# B&R Automation Studio project BenchEDM_AS6 (part 2)

#### TC_IO_AI.st
```iecst
(* Full Analog Input Handler*)
FUNCTION_BLOCK TC_IO_AI

	CASE VarType OF
		TC_IO_ANALOG_TYPE_INT:
		//LOGICAL
			Signal.IOMapping.VarINT					:= IOMapping.VarINT;
			Signal.Vis.Raw							:= INT_TO_LREAL(Signal.IOMapping.VarINT);
			Signal.Vis.IO							:= Par.M*INT_TO_LREAL(Signal.IOMapping.VarINT)+Par.B;
		//SIMULATION
			IF Sim.Active THEN
				Signal.Vis.IO						:= Sim.Logical;
				IF Par.M <> 0 THEN
					Signal.Vis.Raw					:= (Signal.Vis.IO-Par.B)/Par.M;
					Signal.IOMapping.VarINT			:= LREAL_TO_INT(Signal.Vis.Raw);
				ELSE
					Signal.Vis.Raw					:= 0.0;
					Signal.IOMapping.VarINT			:= 0;
				END_IF;
			END_IF;
		TC_IO_ANALOG_TYPE_USINT:
		//LOGICAL
			Signal.IOMapping.VarUSINT				:= IOMapping.VarUSINT;
			Signal.Vis.Raw							:= USINT_TO_LREAL(Signal.IOMapping.VarUSINT);
			Signal.Vis.IO							:= Par.M*USINT_TO_LREAL(Signal.IOMapping.VarUSINT)+Par.B;
		//SIMULATION
			IF Sim.Active THEN
				Signal.Vis.IO						:= Sim.Logical;
				IF Par.M <> 0 THEN
					Signal.Vis.Raw					:= (Signal.Vis.IO-Par.B)/Par.M;
					Signal.IOMapping.VarUSINT		:= LREAL_TO_USINT(Signal.Vis.Raw);
				ELSE
					Signal.Vis.Raw					:= 0.0;
					Signal.IOMapping.VarUSINT		:= 0;
				END_IF;
			END_IF;
		TC_IO_ANALOG_TYPE_SINT:
		//LOGICAL
			Signal.IOMapping.VarSINT				:= IOMapping.VarSINT;
			Signal.Vis.Raw							:= SINT_TO_LREAL(Signal.IOMapping.VarSINT);
			Signal.Vis.IO							:= Par.M*SINT_TO_LREAL(Signal.IOMapping.VarSINT)+Par.B;
		//SIMULATION
			IF Sim.Active THEN
				Signal.Vis.IO						:= Sim.Logical;
				IF Par.M <> 0 THEN
					Signal.Vis.Raw					:= (Signal.Vis.IO-Par.B)/Par.M;
					Signal.IOMapping.VarSINT		:= LREAL_TO_SINT(Signal.Vis.Raw);
				ELSE
					Signal.Vis.Raw					:= 0.0;
					Signal.IOMapping.VarSINT		:= 0;
				END_IF;
			END_IF;
		TC_IO_ANALOG_TYPE_UINT:
		//LOGICAL
			Signal.IOMapping.VarUINT				:= IOMapping.VarUINT;
			Signal.Vis.Raw							:= UINT_TO_LREAL(Signal.IOMapping.VarUINT);
			Signal.Vis.IO							:= Par.M*UINT_TO_LREAL(Signal.IOMapping.VarUINT)+Par.B;
		//SIMULATION
			IF Sim.Active THEN
				Signal.Vis.IO						:= Sim.Logical;
				IF Par.M <> 0 THEN
					Signal.Vis.Raw					:= (Signal.Vis.IO-Par.B)/Par.M;
					Signal.IOMapping.VarUINT		:= LREAL_TO_UINT(Signal.Vis.Raw);
				ELSE
					Signal.Vis.Raw					:= 0.0;
					Signal.IOMapping.VarUINT		:= 0;
				END_IF;
			END_IF;
		TC_IO_ANALOG_TYPE_DINT:
		//LOGICAL
			Signal.IOMapping.VarDINT				:= IOMapping.VarDINT;
			Signal.Vis.Raw							:= DINT_TO_LREAL(Signal.IOMapping.VarDINT);
			Signal.Vis.IO							:= Par.M*DINT_TO_LREAL(Signal.IOMapping.VarDINT)+Par.B;
		//SIMULATION
			IF Sim.Active THEN
				Signal.Vis.IO						:= Sim.Logical;
				IF Par.M <> 0 THEN
					Signal.Vis.Raw					:= (Signal.Vis.IO-Par.B)/Par.M;
					Signal.IOMapping.VarDINT		:= LREAL_TO_DINT(Signal.Vis.Raw);
				ELSE
					Signal.Vis.Raw					:= 0.0;
					Signal.IOMapping.VarDINT		:= 0;
				END_IF;
			END_IF;
		TC_IO_ANALOG_TYPE_UDINT:
		//LOGICAL
			Signal.IOMapping.VarUDINT				:= IOMapping.VarUDINT;
			Signal.Vis.Raw							:= UDINT_TO_LREAL(Signal.IOMapping.VarUDINT);
			Signal.Vis.IO							:= Par.M*UDINT_TO_LREAL(Signal.IOMapping.VarUDINT)+Par.B;
		//SIMULATION
			IF Sim.Active THEN
				Signal.Vis.IO						:= Sim.Logical;
				IF Par.M <> 0 THEN
					Signal.Vis.Raw					:= (Signal.Vis.IO-Par.B)/Par.M;
					Signal.IOMapping.VarUDINT		:= LREAL_TO_UDINT(Signal.Vis.Raw);
				ELSE
					Signal.Vis.Raw					:= 0.0;
					Signal.IOMapping.VarUDINT		:= 0;
				END_IF;
			END_IF;
		TC_IO_ANALOG_TYPE_REAL:
		//LOGICAL
			Signal.IOMapping.VarREAL				:= IOMapping.VarREAL;
			Signal.Vis.Raw							:= REAL_TO_LREAL(Signal.IOMapping.VarREAL);
			Signal.Vis.IO							:= Par.M*REAL_TO_LREAL(Signal.IOMapping.VarREAL)+Par.B;
		//SIMULATION
			IF Sim.Active THEN
				Signal.Vis.IO						:= Sim.Logical;
				IF Par.M <> 0 THEN
					Signal.Vis.Raw					:= (Signal.Vis.IO-Par.B)/Par.M;
					Signal.IOMapping.VarREAL		:= LREAL_TO_REAL(Signal.Vis.Raw);
				ELSE
					Signal.Vis.Raw					:= 0.0;
					Signal.IOMapping.VarREAL		:= 0;
				END_IF;
			END_IF;
		TC_IO_ANALOG_TYPE_LREAL:
		//LOGICAL
			Signal.IOMapping.VarLREAL				:= IOMapping.VarLREAL;
			Signal.Vis.Raw							:= Signal.IOMapping.VarLREAL;
			Signal.Vis.IO							:= Par.M*Signal.IOMapping.VarLREAL+Par.B;
		//SIMULATION
			IF Sim.Active THEN
				Signal.Vis.IO						:= Sim.Logical;
				IF Par.M <> 0 THEN
					Signal.Vis.Raw					:= (Signal.Vis.IO-Par.B)/Par.M;
					Signal.IOMapping.VarLREAL		:= Signal.Vis.Raw;
				ELSE
					Signal.Vis.Raw					:= 0.0;
					Signal.IOMapping.VarLREAL		:= 0;
				END_IF;
			END_IF;
	END_CASE;
	Signal.Logical									:= Signal.Vis.IO;
//FORCING
	IF Forcing.On XOR Forcing.Off THEN
		IF Forcing.Off THEN
			Signal.Logical							:= 0.0;
		ELSIF Forcing.On THEN
			Signal.Logical							:= Forcing.Value;
		END_IF;
	END_IF;
//LIMITING
	Signal.UnlimitedLogical							:= Signal.Logical;
	Signal.MaxExceeded								:= FALSE;
	IF Signal.Logical > Par.MaxValue THEN
		Signal.MaxExceeded							:= TRUE;
		Signal.Logical								:= Par.MaxValue;
	END_IF;
	Signal.MinExceeded								:= FALSE;
	IF Signal.Logical < Par.MinValue THEN
		Signal.MinExceeded							:= TRUE;
		Signal.Logical								:= Par.MinValue;
	END_IF;
//FILTERING
	Internal.Filter 								:= Par.Filter;
	IF Par.Filter < 0.0 THEN
		Internal.Filter 							:= 0.0;
	ELSIF Internal.Filter > 1.0 THEN
		Internal.Filter 							:= 0.99999999;
	END_IF;
	IF NOT Internal.InitFilter OR Internal.LastFilter <> Internal.Filter THEN
		Internal.InitFilter							:= TRUE;
		Internal.LastFilter 						:= Internal.Filter;
		Signal.Filtered 							:= Signal.Logical;
	ELSE
		Signal.Filtered 							:= Signal.Logical*(1.0-Internal.Filter) + Signal.Filtered*Internal.Filter;
	END_IF;
	IF Signal.Filtered > Par.MaxValue THEN
		Signal.Filtered 							:= Par.MaxValue;
	ELSIF Signal.Filtered < Par.MinValue THEN
		Signal.Filtered 							:= Par.MinValue;
	END_IF;
	Signal.Vis.App									:= Signal.Filtered;
END_FUNCTION_BLOCK
```

### Library Logical/Libraries/TC_Dir (IEC)
Depends on: TC_General, AsBrStr, standard, brsystem, FileIO, AsUSB, astime

#### Types.typ - Exported data types
```iecst
TYPE
	TC_DirDef_Sanitize_typ : 	STRUCT
		AllowUndefinedDir : BOOL;
		SanitizeFilesByExt : BOOL;
		SanitizeFilesByRoot : BOOL;
		FileExtension : STRING[260];
		FileRoot : STRING[260];
		MaxSize : UDINT;
		MaxFiles : UDINT;
	END_STRUCT;
	TC_DirDef_typ : 	STRUCT
		Valid : BOOL;
		DirPath : STRING[260];
		Sanitize : TC_DirDef_Sanitize_typ;
	END_STRUCT;
	TC_DirMake_Internal_typ : 	STRUCT
		State : TC_DIRMAKE_STATE_ENUM;
		DirDefItem : TC_DirDef_typ;
		DirCreate_0 : DirCreate;
		DirIdx : INT;
	END_STRUCT;
	TC_DIRMAKE_STATE_ENUM :
		(
		DIRMAKE_RESET,
		DIRMAKE_IDLE,
		DIRMAKE_CREATE_CMD,
		DIRMAKE_CREATE_WAIT,
		DIRMAKE_DONE,
		DIRMAKE_ERROR
		);
	TC_DirReadAll_Internal_typ : 	STRUCT
		State : TC_DIRREADALL_STATE_ENUM;
		DirOpen_0 : DirOpen;
		DirReadEx_0 : DirReadEx;
		DirClose_0 : DirClose;
		i : INT;
		FileListIdx : INT;
		DirIdent : UDINT;
		DirData : fiDIR_READ_EX_DATA;
		FileListItem : TC_FileList_typ;
		CurrentDirPath : STRING[260];
	END_STRUCT;
	TC_DIRREADALL_STATE_ENUM :
		(
		DIRREADALL_RESET,
		DIRREADALL_IDLE,
		DIRREADALL_OPEN_CMD,
		DIRREADALL_OPEN_WAIT,
		DIRREADALL_READ_CMD,
		DIRREADALL_READ_WAIT,
		DIRREADALL_CLOSE_WAIT,
		DIRREADALL_EVALUATE,
		DIRREADALL_DONE,
		DIRREADALL_ERROR
		);
	TC_DirSanitize_Internal_typ : 	STRUCT
		State : TC_DIRSANITIZE_STATE_ENUM;
		DirDeleteEx_0 : DirDeleteEx;
		FileDelete_0 : FileDelete;
		DirDefItem : TC_DirDef_typ;
		FileListItem : TC_FileList_typ;
		FileListItem1 : TC_FileList_typ;
		i : INT;
		j : INT;
		FileListIdx : INT;
		Size : UDINT;
		DirIdent : UDINT;
		SizeCount : UDINT;
		FileCount : UDINT;
		DirData : fiDIR_READ_EX_DATA;
		Found : BOOL;
		Find : INT;
		TempPath : STRING[260];
		CurrentDirIdx : INT;
	END_STRUCT;
	TC_DIRSANITIZE_STATE_ENUM :
		(
		DIRSANITIZE_RESET,
		DIRSANITIZE_IDLE,
		DIRSANITIZE_EVALUATE_DIR,
		DIRSANITIZE_DELETE_DIR_CMD,
		DIRSANITIZE_DELETE_DIR_WAIT,
		DIRSANITIZE_DELETE_DIR_PROCESS,
		DIRSANITIZE_EVALUATE_FILE,
		DIRSANITIZE_DELETE_FILE_CMD,
		DIRSANITIZE_DELETE_FILE_WAIT,
		DIRSANITIZE_DONE,
		DIRSANITIZE_ERROR
		);
	TC_Dir_Transfer_Internal_typ : 	STRUCT
		State : TC_DIR_TRANSFER_STATE_ENUM;
		TransferListItem : TC_Dir_Transfer_List_typ;
		ListIdx : INT;
		DirCopy_0 : DirCopy;
		FileCopy_0 : FileCopy;
		DirDeleteEx_0 : DirDeleteEx;
		DirCreate_0 : DirCreate;
		FileDelete_0 : FileDelete;
	END_STRUCT;
	TC_Dir_Transfer_List_typ : 	STRUCT
		Valid : BOOL;
		SrcOrDestUSB : BOOL;
		IsDir : BOOL;
		SrcDelete : BOOL;
		SrcCreateDir : BOOL;
		NoTransfer : BOOL;
		SrcDev : STRING[80];
		SrcPath : STRING[260];
		DestDev : STRING[80];
		DestPath : STRING[260];
	END_STRUCT;
	TC_DIR_TRANSFER_STATE_ENUM :
		(
		TRANSFER_RESET,
		TRANSFER_IDLE,
		TRANSFER_CHECK_LIST,
		TRANSFER_DIR_COPY_CMD,
		TRANSFER_DIR_COPY_WAIT,
		TRANSFER_FILE_COPY_CMD,
		TRANSFER_FILE_COPY_WAIT,
		TRANSFER_DIR_DELETE_CMD,
		TRANSFER_DIR_DELETE_WAIT,
		TRANSFER_FILE_DELETE_CMD,
		TRANSFER_FILE_DELETE_WAIT,
		TRANSFER_DIR_CREATE_CMD,
		TRANSFER_DIR_CREATE_WAIT,
		TRANSFER_DONE,
		TRANSFER_ERROR
		);
	TC_Dir_USB_Connect_Internal_typ : 	STRUCT
		UsbNodeListGet_0 : UsbNodeListGet;
		UsbNodeGet_0 : UsbNodeGet;
		DevLink_0 : DevLink;
		UsbMsDeviceReady_0 : UsbMsDeviceReady;
		DevUnlink_0 : DevUnlink;
		CTON_Delay : CTON;
		NodeList : UDINT;
		Node : usbNode_typ;
		ParString : STRING[1000];
		Handle : UDINT;
		State : TC_USB_CONNECT_STATE_ENUM;
	END_STRUCT;
	TC_FileList_typ : 	STRUCT
		Path : STRING[260];
		DateUDINT : UDINT;
		Size : UDINT;
		IsDir : BOOL;
		DirIdx : INT;
		Internal : USINT; (*0=unread, 1=delete, 2=parentDirDelete, 3=remove*)
	END_STRUCT;
	TC_USB_CONNECT_STATE_ENUM :
		(
		USB_CONNECT_RESET,
		USB_CONNECT_IDLE,
		USB_CONNECT_GET_LIST_CMD,
		USB_CONNECT_GET_LIST_WAIT,
		USB_CONNECT_GET_NODE_CMD,
		USB_CONNECT_GET_NODE_WAIT,
		USB_CONNECT_DEVLINK_CMD,
		USB_CONNECT_DEVLINK_WAIT,
		USB_CONNECT_CHECK_CONNECTED,
		USB_CONNECT_CONNECTED,
		USB_CONNECT_DEVUNLINK_CMD,
		USB_CONNECT_DEVUNLINK_WAIT,
		USB_CONNECT_DELAY,
		USB_CONNECT_DONE,
		USB_CONNECT_ERROR
		);
END_TYPE
```

#### TC_Dir.fun - Exported functions and function blocks
```iecst
{REDUND_ERROR} FUNCTION_BLOCK TC_DirMake (* *) (*$GROUP=User,$CAT=User,$GROUPICON=User.png,$CATICON=User.png*)
	VAR_INPUT
		enable : BOOL;
		pDevice : UDINT;
		pDirDef : UDINT;
	END_VAR
	VAR_OUTPUT
		status : UINT;
	END_VAR
	VAR
		Internal : TC_DirMake_Internal_typ;
	END_VAR
END_FUNCTION_BLOCK

{REDUND_ERROR} FUNCTION_BLOCK TC_DirReadAll (*Reads Entire File Device*) (*$GROUP=User,$CAT=User,$GROUPICON=User.png,$CATICON=User.png*)
	VAR_INPUT
		enable : BOOL;
		pDevice : UDINT;
		pFileList : UDINT;
	END_VAR
	VAR_OUTPUT
		status : UINT;
	END_VAR
	VAR
		Internal : TC_DirReadAll_Internal_typ;
	END_VAR
END_FUNCTION_BLOCK

{REDUND_ERROR} FUNCTION_BLOCK TC_DirSanitize (*Sanitizes File Device*) (*$GROUP=User,$CAT=User,$GROUPICON=User.png,$CATICON=User.png*)
	VAR_INPUT
		enable : BOOL;
		pDevice : UDINT;
		pDirDef : UDINT;
		pFileList : UDINT;
	END_VAR
	VAR_OUTPUT
		status : UINT;
	END_VAR
	VAR
		Internal : TC_DirSanitize_Internal_typ;
	END_VAR
END_FUNCTION_BLOCK

{REDUND_ERROR} FUNCTION_BLOCK TC_Dir_USB_Connect (*TODO: Add your comment here*) (*$GROUP=User,$CAT=User,$GROUPICON=User.png,$CATICON=User.png*)
	VAR_INPUT
		enable : BOOL;
		reset : BOOL;
		refresh : BOOL;
		delay : REAL;
	END_VAR
	VAR_OUTPUT
		status : UINT;
		connected : BOOL;
	END_VAR
	VAR
		Internal : TC_Dir_USB_Connect_Internal_typ;
	END_VAR
END_FUNCTION_BLOCK

{REDUND_ERROR} FUNCTION_BLOCK TC_Dir_Transfer (*Transfer List from Device to Another*) (*$GROUP=User,$CAT=User,$GROUPICON=User.png,$CATICON=User.png*)
	VAR_INPUT
		enable : BOOL;
		USB_Connected : BOOL;
		pTransferList : UDINT;
	END_VAR
	VAR_OUTPUT
		index : INT;
		status : UINT;
	END_VAR
	VAR
		Internal : TC_Dir_Transfer_Internal_typ;
	END_VAR
END_FUNCTION_BLOCK
```

#### TC_DirMake.st
```iecst
FUNCTION_BLOCK TC_DirMake

	IF enable = FALSE THEN
		Internal.State									:= DIRMAKE_RESET;
	END_IF;

	CASE Internal.State OF
		DIRMAKE_RESET:
			status										:= 65534;
			brsmemset(ADR(Internal),0,SIZEOF(Internal));
			Internal.State								:= DIRMAKE_IDLE;
		DIRMAKE_IDLE:
			status										:= 65534;
			IF enable THEN
				IF pDevice <> 0 AND pDirDef <> 0 THEN
					status								:= 65535;
					brsmemset(ADR(Internal),0,SIZEOF(Internal));
					Internal.State						:= DIRMAKE_CREATE_CMD;
				ELSE
					status								:= 60001;
					Internal.State						:= DIRMAKE_ERROR;
				END_IF;
			END_IF;
		DIRMAKE_CREATE_CMD:
			status										:= 65535;
			IF Internal.DirIdx >= 0 AND Internal.DirIdx <= MAX_DIR_DEF_IDX THEN
				brsmemcpy(ADR(Internal.DirDefItem),pDirDef+SIZEOF(Internal.DirDefItem)*Internal.DirIdx,SIZEOF(Internal.DirDefItem));
				IF Internal.DirDefItem.Valid THEN
					IF Internal.DirDefItem.DirPath <> '' AND Internal.DirDefItem.DirPath <> '/' THEN
						Internal.DirCreate_0.enable 	:= TRUE;
						Internal.DirCreate_0.pDevice	:= pDevice;
						Internal.DirCreate_0.pName		:= ADR(Internal.DirDefItem.DirPath);
						Internal.State					:= DIRMAKE_CREATE_WAIT;
					ELSE
						Internal.DirIdx 				:= Internal.DirIdx + 1;
					END_IF;
				ELSE
					Internal.State						:= DIRMAKE_DONE;
				END_IF;
			ELSE
				Internal.State							:= DIRMAKE_DONE;
			END_IF;
		DIRMAKE_CREATE_WAIT:
			status										:= 65535;
			IF Internal.DirCreate_0.status = ERR_OK OR Internal.DirCreate_0.status = fiERR_DIR_ALREADY_EXIST THEN
				Internal.DirCreate_0.enable 			:= FALSE;
				Internal.DirIdx 						:= Internal.DirIdx + 1;
				Internal.State 							:= DIRMAKE_CREATE_CMD;
			ELSIF Internal.DirCreate_0.status <> ERR_FUB_BUSY AND Internal.DirCreate_0.status <> ERR_FUB_ENABLE_FALSE THEN
				Internal.DirCreate_0.enable 			:= FALSE;
				status									:= Internal.DirCreate_0.status;
				Internal.State 							:= DIRMAKE_ERROR;
			END_IF;
		DIRMAKE_DONE:
			status										:= 0;
		DIRMAKE_ERROR:
			// Error
	END_CASE;
	Internal.DirCreate_0();

END_FUNCTION_BLOCK
```

#### TC_DirSanitize.st
```iecst
(* Sanitizes File Device *)
FUNCTION_BLOCK TC_DirSanitize
	IF enable = FALSE THEN
		Internal.State										:= DIRSANITIZE_RESET;
	END_IF;

	CASE Internal.State OF
		DIRSANITIZE_RESET:
			status											:= 65534;
			brsmemset(ADR(Internal),0,SIZEOF(Internal));
			Internal.State									:= DIRSANITIZE_IDLE;
		DIRSANITIZE_IDLE:
			status											:= 65534;
			IF enable THEN
				IF pDevice <> 0 AND pDirDef <> 0 AND pFileList <> 0 THEN
					brsmemset(ADR(Internal),0,SIZEOF(Internal));
					status									:= 65535;
					Internal.State							:= DIRSANITIZE_EVALUATE_DIR;
				ELSE
					brsmemset(ADR(Internal),0,SIZEOF(Internal));
					status									:= 60001;
					Internal.State							:= DIRSANITIZE_ERROR;
				END_IF;
			END_IF;
		DIRSANITIZE_EVALUATE_DIR:
			status											:= 65535;
			// Determine DirIdx
			FOR Internal.i := 0 TO MAX_DIR_MAN_FILE_LIST_IDX DO
				brsmemcpy(ADR(Internal.FileListItem),pFileList+SIZEOF(Internal.FileListItem)*Internal.i,SIZEOF(Internal.FileListItem));
				IF Internal.FileListItem.Path = '' AND Internal.FileListItem.IsDir = FALSE THEN
					EXIT;
				ELSE
					Internal.Found 							:= FALSE;
					FOR Internal.j := 0 TO MAX_DIR_DEF_IDX DO
						brsmemcpy(ADR(Internal.DirDefItem),pDirDef+SIZEOF(Internal.DirDefItem)*Internal.j,SIZEOF(Internal.DirDefItem));
						IF Internal.DirDefItem.Valid THEN
							IF Internal.FileListItem.Path = Internal.DirDefItem.DirPath OR Internal.FileListItem.Path = '' THEN
								Internal.FileListItem.DirIdx := Internal.j;
								Internal.Found 				:= TRUE;
								EXIT;
							END_IF;
						END_IF;
					END_FOR;
					IF NOT Internal.Found THEN
						FOR Internal.j := MAX_DIR_DEF_IDX TO 0 BY -1 DO
							brsmemcpy(ADR(Internal.DirDefItem),pDirDef+SIZEOF(Internal.DirDefItem)*Internal.j,SIZEOF(Internal.DirDefItem));
							IF Internal.DirDefItem.Valid THEN
								Internal.Find := FIND(Internal.FileListItem.Path,Internal.DirDefItem.DirPath);
								IF Internal.Find <> 0 THEN
									Internal.TempPath := DELETE(Internal.FileListItem.Path,LEN(Internal.DirDefItem.DirPath),1);
									IF FIND(Internal.TempPath,'/') <> 0 OR Internal.DirDefItem.DirPath = '' THEN
										Internal.FileListItem.DirIdx := Internal.j;
										EXIT;
									END_IF;
								END_IF;
							END_IF;
						END_FOR;
					END_IF;
					brsmemcpy(pFileList+SIZEOF(Internal.FileListItem)*Internal.i,ADR(Internal.FileListItem),SIZEOF(Internal.FileListItem));
				END_IF;
			END_FOR;

			// Handle Directory Sanitation
			Internal.Found									:= FALSE;
			FOR Internal.i := 0 TO MAX_DIR_MAN_FILE_LIST_IDX DO
				brsmemcpy(ADR(Internal.FileListItem),pFileList+SIZEOF(Internal.FileListItem)*Internal.i,SIZEOF(Internal.FileListItem));
				IF Internal.FileListItem.Path = '' AND Internal.FileListItem.IsDir = FALSE THEN
					EXIT;
				ELSIF Internal.FileListItem.IsDir THEN
					brsmemcpy(ADR(Internal.DirDefItem),pDirDef+SIZEOF(Internal.DirDefItem)*Internal.FileListItem.DirIdx,SIZEOF(Internal.DirDefItem));
					IF NOT Internal.DirDefItem.Sanitize.AllowUndefinedDir AND Internal.DirDefItem.DirPath <> Internal.FileListItem.Path THEN
						Internal.Found					:= TRUE;
						Internal.FileListItem.Internal.1 := 1;
						brsmemcpy(pFileList+SIZEOF(Internal.FileListItem)*Internal.i,ADR(Internal.FileListItem),SIZEOF(Internal.FileListItem));
					END_IF;
				END_IF;
			END_FOR;
			Internal.State 									:= DIRSANITIZE_DELETE_DIR_CMD;
		DIRSANITIZE_DELETE_DIR_CMD:
			status											:= 65535;
			Internal.Found									:= FALSE;
			FOR Internal.i := 0 TO MAX_DIR_MAN_FILE_LIST_IDX DO
				brsmemcpy(ADR(Internal.FileListItem),pFileList+SIZEOF(Internal.FileListItem)*Internal.i,SIZEOF(Internal.FileListItem));
				IF Internal.FileListItem.Path = '' AND Internal.FileListItem.IsDir = FALSE THEN
					EXIT;
				ELSIF Internal.FileListItem.IsDir AND Internal.FileListItem.Internal.1 = 1 AND NOT Internal.FileListItem.Internal.2 = 1 THEN
					Internal.Found							:= TRUE;
					EXIT;
				END_IF;
			END_FOR;
			IF Internal.Found THEN
				Internal.DirDeleteEx_0.enable 				:= TRUE;
				Internal.DirDeleteEx_0.pDevice 				:= pDevice;
				Internal.DirDeleteEx_0.pName 				:= ADR(Internal.FileListItem.Path);
				Internal.State 								:= DIRSANITIZE_DELETE_DIR_WAIT;
			ELSE
				Internal.State 								:= DIRSANITIZE_EVALUATE_FILE;
			END_IF;
		DIRSANITIZE_DELETE_DIR_WAIT:
			status											:= 65535;
			IF Internal.DirDeleteEx_0.status = 0 OR (Internal.DirDeleteEx_0.status <> ERR_FUB_BUSY AND Internal.DirDeleteEx_0.status <> ERR_FUB_ENABLE_FALSE) THEN
				Internal.DirDeleteEx_0.enable 				:= FALSE;
				Internal.FileListItem1 						:= Internal.FileListItem;
				FOR Internal.i := 0 TO MAX_DIR_MAN_FILE_LIST_IDX DO
					brsmemcpy(ADR(Internal.FileListItem),pFileList+SIZEOF(Internal.FileListItem)*Internal.i,SIZEOF(Internal.FileListItem));
					IF Internal.FileListItem.Path = '' AND Internal.FileListItem.IsDir = FALSE THEN
						EXIT;
					ELSIF FIND(Internal.FileListItem.Path,Internal.FileListItem1.Path) <> 0 THEN
						Internal.FileListItem.Internal.3 	:= 1;
						brsmemcpy(pFileList+SIZEOF(Internal.FileListItem)*Internal.i,ADR(Internal.FileListItem),SIZEOF(Internal.FileListItem));
					END_IF;
				END_FOR;
				Internal.j 									:= 0;
				FOR Internal.i := 0 TO MAX_DIR_MAN_FILE_LIST_IDX DO
					brsmemcpy(ADR(Internal.FileListItem),pFileList+SIZEOF(Internal.FileListItem)*Internal.i,SIZEOF(Internal.FileListItem));
					IF Internal.FileListItem.Path = '' AND Internal.FileListItem.IsDir = FALSE THEN
						EXIT;
					ELSIF Internal.FileListItem.Internal.3 = 0 THEN
						IF Internal.j <> Internal.i THEN
							Internal.Size						:= (MAX_DIR_MAN_FILE_LIST_IDX+1-Internal.i);
							brsmemmove(pFileList+Internal.j*SIZEOF(Internal.FileListItem),pFileList+Internal.i*SIZEOF(Internal.FileListItem),SIZEOF(Internal.FileListItem)*Internal.Size);
							brsmemset(pFileList+(Internal.j+Internal.Size)*SIZEOF(Internal.FileListItem),0,SIZEOF(Internal.FileListItem)*(Internal.i-Internal.j));
						END_IF;
						Internal.j							:= Internal.j + (Internal.i-Internal.j)+1;
						Internal.i							:= Internal.j-1;
					ELSE
						brsmemset(pFileList+Internal.i*SIZEOF(Internal.FileListItem),0,SIZEOF(Internal.FileListItem));
					END_IF;
				END_FOR;
				Internal.State 								:= DIRSANITIZE_DELETE_DIR_CMD;
			END_IF;
		DIRSANITIZE_EVALUATE_FILE:
			status											:= 65535;

			// Handle File Sanitation By Root
			Internal.Found									:= FALSE;
			FOR Internal.i := 0 TO MAX_DIR_MAN_FILE_LIST_IDX DO
				brsmemcpy(ADR(Internal.FileListItem),pFileList+SIZEOF(Internal.FileListItem)*Internal.i,SIZEOF(Internal.FileListItem));
				IF Internal.FileListItem.Path = '' AND Internal.FileListItem.IsDir = FALSE THEN
					EXIT;
				ELSIF NOT Internal.FileListItem.IsDir THEN
					brsmemcpy(ADR(Internal.DirDefItem),pDirDef+SIZEOF(Internal.DirDefItem)*Internal.FileListItem.DirIdx,SIZEOF(Internal.DirDefItem));
					IF Internal.DirDefItem.Sanitize.SanitizeFilesByRoot THEN
						Internal.TempPath 					:= '';
						brsstrcat(ADR(Internal.TempPath),ADR(Internal.DirDefItem.DirPath));
						brsstrcat(ADR(Internal.TempPath),ADR('/'));
						brsstrcat(ADR(Internal.TempPath),ADR(Internal.DirDefItem.Sanitize.FileRoot));
						IF FIND(Internal.FileListItem.Path,Internal.TempPath) = 0 THEN
							Internal.Found					:= TRUE;
							Internal.FileListItem.Internal.1 := 1;
							brsmemcpy(pFileList+SIZEOF(Internal.FileListItem)*Internal.i,ADR(Internal.FileListItem),SIZEOF(Internal.FileListItem));
						END_IF;
					END_IF;
					IF Internal.DirDefItem.Sanitize.SanitizeFilesByExt THEN
						IF FIND(Internal.FileListItem.Path,Internal.DirDefItem.Sanitize.FileExtension) = 0 THEN
							Internal.Found					:= TRUE;
							Internal.FileListItem.Internal.1 := 1;
							brsmemcpy(pFileList+SIZEOF(Internal.FileListItem)*Internal.i,ADR(Internal.FileListItem),SIZEOF(Internal.FileListItem));
						END_IF;
					END_IF;
				END_IF;
			END_FOR;

			// Check if found in the last step. If so we have to go delete these files before counting them for size and number of files.
			IF Internal.Found THEN
				Internal.State 								:= DIRSANITIZE_DELETE_FILE_CMD;
			ELSE
				// Reorder Files for Evaluation
				FOR Internal.i := 0 TO MAX_DIR_MAN_FILE_LIST_IDX-1 DO
					brsmemcpy(ADR(Internal.FileListItem),pFileList+SIZEOF(Internal.FileListItem)*Internal.i,SIZEOF(Internal.FileListItem));
					brsmemcpy(ADR(Internal.FileListItem1),pFileList+SIZEOF(Internal.FileListItem1)*(Internal.i+1),SIZEOF(Internal.FileListItem1));
					IF (Internal.FileListItem.Path = '' AND Internal.FileListItem.IsDir = FALSE) OR (Internal.FileListItem1.Path = '' AND Internal.FileListItem1.IsDir = FALSE) THEN
						EXIT;
					ELSE
						IF Internal.FileListItem.DirIdx = Internal.FileListItem1.DirIdx THEN
							IF Internal.FileListItem.DateUDINT < Internal.FileListItem1.DateUDINT THEN
								brsmemcpy(pFileList+SIZEOF(Internal.FileListItem1)*Internal.i,ADR(Internal.FileListItem1),SIZEOF(Internal.FileListItem1));
								brsmemcpy(pFileList+SIZEOF(Internal.FileListItem)*(Internal.i+1),ADR(Internal.FileListItem),SIZEOF(Internal.FileListItem));
							END_IF;
						END_IF;
					END_IF;
				END_FOR;
				// Delete Files Based On File Number and Size Restriction
				Internal.Found								:= FALSE;
				Internal.CurrentDirIdx						:= 0;
				Internal.FileCount							:= 1;
				Internal.SizeCount							:= 0;
				FOR Internal.i := 0 TO MAX_DIR_MAN_FILE_LIST_IDX DO
					brsmemcpy(ADR(Internal.FileListItem),pFileList+SIZEOF(Internal.FileListItem)*Internal.i,SIZEOF(Internal.FileListItem));
					IF Internal.FileListItem.Path = '' AND Internal.FileListItem.IsDir = FALSE THEN
						EXIT;
					ELSIF NOT Internal.FileListItem.IsDir THEN
						IF Internal.CurrentDirIdx <> Internal.FileListItem.DirIdx THEN
							Internal.CurrentDirIdx 			:= Internal.FileListItem.DirIdx;
							Internal.FileCount				:= 1;
							Internal.SizeCount				:= Internal.FileListItem.Size;
						ELSE
							Internal.FileCount				:= Internal.FileCount + 1;
							Internal.SizeCount				:= Internal.SizeCount + Internal.FileListItem.Size;
						END_IF;
						brsmemcpy(ADR(Internal.DirDefItem),pDirDef+SIZEOF(Internal.DirDefItem)*Internal.FileListItem.DirIdx,SIZEOF(Internal.DirDefItem));
						IF Internal.FileCount > Internal.DirDefItem.Sanitize.MaxFiles OR Internal.SizeCount > Internal.DirDefItem.Sanitize.MaxSize THEN
							Internal.Found					:= TRUE;
							Internal.FileListItem.Internal.1 := 1;
							brsmemcpy(pFileList+SIZEOF(Internal.FileListItem)*Internal.i,ADR(Internal.FileListItem),SIZEOF(Internal.FileListItem));
						END_IF;
					END_IF;
				END_FOR;
				IF Internal.Found THEN
					Internal.State 							:= DIRSANITIZE_DELETE_FILE_CMD;
				ELSE
					Internal.State 							:= DIRSANITIZE_DONE;
				END_IF;
			END_IF;
		DIRSANITIZE_DELETE_FILE_CMD:
			status											:= 65535;
			Internal.Found									:= FALSE;
			FOR Internal.i := 0 TO MAX_DIR_MAN_FILE_LIST_IDX DO
				brsmemcpy(ADR(Internal.FileListItem),pFileList+SIZEOF(Internal.FileListItem)*Internal.i,SIZEOF(Internal.FileListItem));
				IF Internal.FileListItem.Path = '' AND Internal.FileListItem.IsDir = FALSE THEN
					EXIT;
				ELSIF NOT Internal.FileListItem.IsDir AND Internal.FileListItem.Internal.1 = 1 THEN
					Internal.FileListItem.Internal.1 := 0;
					Internal.FileListItem.Internal.3 := 1;
					brsmemcpy(pFileList+SIZEOF(Internal.FileListItem)*Internal.i,ADR(Internal.FileListItem),SIZEOF(Internal.FileListItem));
					Internal.Found							:= TRUE;
					EXIT;
				END_IF;
			END_FOR;
			IF Internal.Found THEN
				Internal.FileDelete_0.enable 				:= TRUE;
				Internal.FileDelete_0.pDevice 				:= pDevice;
				Internal.FileDelete_0.pName 				:= ADR(Internal.FileListItem.Path);
				Internal.State 								:= DIRSANITIZE_DELETE_FILE_WAIT;
			ELSE
				Internal.State 								:= DIRSANITIZE_EVALUATE_FILE;
			END_IF;
		DIRSANITIZE_DELETE_FILE_WAIT:
			status											:= 65535;
			IF Internal.FileDelete_0.status = 0 OR (Internal.FileDelete_0.status <> ERR_FUB_BUSY AND Internal.FileDelete_0.status <> ERR_FUB_ENABLE_FALSE) THEN
				Internal.FileDelete_0.enable 				:= FALSE;
				Internal.j 									:= 0;
				FOR Internal.i := 0 TO MAX_DIR_MAN_FILE_LIST_IDX DO
					brsmemcpy(ADR(Internal.FileListItem),pFileList+SIZEOF(Internal.FileListItem)*Internal.i,SIZEOF(Internal.FileListItem));
					IF Internal.FileListItem.Path = '' AND Internal.FileListItem.IsDir = FALSE THEN
						EXIT;
					ELSIF Internal.FileListItem.Internal.3 = 0 THEN
						IF Internal.j <> Internal.i THEN
							Internal.Size						:= (MAX_DIR_MAN_FILE_LIST_IDX+1-Internal.i);
							brsmemmove(pFileList+Internal.j*SIZEOF(Internal.FileListItem),pFileList+Internal.i*SIZEOF(Internal.FileListItem),SIZEOF(Internal.FileListItem)*Internal.Size);
							brsmemset(pFileList+(Internal.j+Internal.Size)*SIZEOF(Internal.FileListItem),0,SIZEOF(Internal.FileListItem)*(Internal.i-Internal.j));
						END_IF;
						Internal.j							:= Internal.j + (Internal.i-Internal.j)+1;
						Internal.i							:= Internal.j-1;
					ELSE
						brsmemset(pFileList+Internal.i*SIZEOF(Internal.FileListItem),0,SIZEOF(Internal.FileListItem));
					END_IF;
				END_FOR;
				Internal.State 								:= DIRSANITIZE_DELETE_FILE_CMD;
			END_IF;
		DIRSANITIZE_DONE:
			status											:= 0;
		DIRSANITIZE_ERROR:
			// Error
	END_CASE;

	Internal.FileDelete_0();
	Internal.DirDeleteEx_0();

END_FUNCTION_BLOCK
```

#### TC_Dir_USB_Connect.st
```iecst
// This function only supports a single USB flash drive, additional will be ignored.
// When connected the USB can be accessed using Dev Name 'USB_DEVICE'

FUNCTION_BLOCK TC_Dir_USB_Connect

	IF enable = FALSE OR reset THEN
		Internal.State											:= USB_CONNECT_RESET;
	END_IF;

	CASE Internal.State OF
		USB_CONNECT_RESET:
			status												:= 65534;
			brsmemset(ADR(Internal),0,SIZEOF(Internal));
			connected											:= FALSE;
			Internal.State										:= USB_CONNECT_IDLE;
		USB_CONNECT_IDLE:
			status												:= 65534;
			IF enable THEN
				status											:= 65535;
				Internal.State									:= USB_CONNECT_GET_LIST_CMD;
			END_IF;
		USB_CONNECT_GET_LIST_CMD:
			status												:= 65535;
			Internal.UsbNodeListGet_0.enable 					:= TRUE;
			Internal.UsbNodeListGet_0.pBuffer 					:= ADR(Internal.NodeList);
			Internal.UsbNodeListGet_0.bufferSize 				:= SIZEOF(Internal.NodeList);
			Internal.UsbNodeListGet_0.filterInterfaceClass 		:= 8; // FIND ONLY USB FLASH DRIVES
			Internal.UsbNodeListGet_0.filterInterfaceSubClass 	:= 6; // FIND ONLY USB FLASH DRIVES
			Internal.State 										:= USB_CONNECT_GET_LIST_WAIT;
		USB_CONNECT_GET_LIST_WAIT:
			status												:= 65535;
			IF Internal.UsbNodeListGet_0.status = 0 THEN
				Internal.UsbNodeListGet_0.enable 				:= FALSE;
				Internal.State 									:= USB_CONNECT_GET_NODE_CMD;
			ELSIF Internal.UsbNodeListGet_0.status <> ERR_FUB_BUSY AND Internal.UsbNodeListGet_0.status <> ERR_FUB_ENABLE_FALSE THEN
				IF Internal.UsbNodeListGet_0.status <> asusbERR_USB_NOTFOUND THEN
					Internal.UsbNodeListGet_0.enable 			:= FALSE;
					status										:= Internal.UsbNodeListGet_0.status;
					Internal.State 								:= USB_CONNECT_ERROR;
				ELSE
					Internal.UsbNodeListGet_0.enable 			:= FALSE;
					Internal.State 								:= USB_CONNECT_DELAY;
				END_IF;
			END_IF;
		USB_CONNECT_GET_NODE_CMD:
			status												:= 65535;
			Internal.UsbNodeGet_0.enable 						:= TRUE;
			Internal.UsbNodeGet_0.pBuffer 						:= ADR(Internal.Node);
			Internal.UsbNodeGet_0.bufferSize 					:= SIZEOF(Internal.Node);
			Internal.UsbNodeGet_0.nodeId 						:= Internal.NodeList;
			Internal.State 										:= USB_CONNECT_GET_NODE_WAIT;
		USB_CONNECT_GET_NODE_WAIT:
			status												:= 65535;
			IF Internal.UsbNodeGet_0.status = 0 THEN
				Internal.UsbNodeGet_0.enable 					:= FALSE;
				brsmemset(ADR(Internal.ParString),0,SIZEOF(Internal.ParString));
				brsstrcat(ADR(Internal.ParString),ADR('/DEVICE='));
				brsstrcat(ADR(Internal.ParString), ADR(Internal.Node.ifName));
				Internal.State 									:= USB_CONNECT_DEVLINK_CMD;
			ELSIF Internal.UsbNodeGet_0.status <> ERR_FUB_BUSY AND Internal.UsbNodeGet_0.status <> ERR_FUB_ENABLE_FALSE THEN
				IF Internal.UsbNodeGet_0.status <> asusbERR_USB_NOTFOUND THEN
					Internal.UsbNodeGet_0.enable 				:= FALSE;
					status										:= Internal.UsbNodeGet_0.status;
					Internal.State 								:= USB_CONNECT_ERROR;
				ELSE
					Internal.UsbNodeGet_0.enable 				:= FALSE;
					Internal.State 								:= USB_CONNECT_DELAY;
				END_IF;
			END_IF;
		USB_CONNECT_DEVLINK_CMD:
			status												:= 65535;
			Internal.DevLink_0.enable 							:= TRUE;
			Internal.DevLink_0.pDevice 							:= ADR('USB_DEVICE');
			Internal.DevLink_0.pParam 							:= ADR(Internal.ParString);
			Internal.State 										:= USB_CONNECT_DEVLINK_WAIT;
		USB_CONNECT_DEVLINK_WAIT:
			status												:= 65535;
			IF Internal.DevLink_0.status = 0 THEN
				Internal.DevLink_0.enable 						:= FALSE;
				Internal.Handle									:= Internal.DevLink_0.handle;
				connected										:= FALSE;
				Internal.State 									:= USB_CONNECT_CHECK_CONNECTED;
			ELSIF Internal.DevLink_0.status <> ERR_FUB_BUSY AND Internal.DevLink_0.status <> ERR_FUB_ENABLE_FALSE THEN
				Internal.DevLink_0.enable 						:= FALSE;
				Internal.State 									:= USB_CONNECT_DEVUNLINK_CMD;
			END_IF;
		USB_CONNECT_CHECK_CONNECTED:
			status												:= 65535;
			Internal.UsbMsDeviceReady_0.enable					:= TRUE;
			Internal.UsbMsDeviceReady_0.pIfName					:= ADR(Internal.Node.ifName);
			Internal.State 										:= USB_CONNECT_CONNECTED;
		USB_CONNECT_CONNECTED:
			status												:= 65535;
			IF Internal.UsbMsDeviceReady_0.status = 0 THEN
				connected										:= TRUE;
				Internal.UsbMsDeviceReady_0.enable 				:= FALSE;
				Internal.State 									:= USB_CONNECT_CHECK_CONNECTED;
			ELSIF Internal.UsbMsDeviceReady_0.status <> ERR_FUB_BUSY AND Internal.UsbMsDeviceReady_0.status <> ERR_FUB_ENABLE_FALSE THEN
				Internal.UsbMsDeviceReady_0.enable 				:= FALSE;
				Internal.State 									:= USB_CONNECT_DEVUNLINK_CMD;
			END_IF;
		USB_CONNECT_DEVUNLINK_CMD:
			status												:= 65535;
			Internal.DevUnlink_0.enable 						:= TRUE;
			Internal.DevUnlink_0.handle 						:= Internal.Handle;
			Internal.State 										:= USB_CONNECT_DEVUNLINK_WAIT;
		USB_CONNECT_DEVUNLINK_WAIT:
			status												:= 65535;
			IF Internal.DevUnlink_0.status = 0 OR (Internal.DevUnlink_0.status <> ERR_FUB_BUSY AND Internal.DevUnlink_0.status <> ERR_FUB_ENABLE_FALSE) THEN
				Internal.DevUnlink_0.enable 					:= FALSE;
				Internal.State 									:= USB_CONNECT_DELAY;
			END_IF;
		USB_CONNECT_DELAY:
			status												:= 65535;
			IF Internal.CTON_Delay.Q OR refresh THEN
				refresh 										:= FALSE;
				Internal.CTON_Delay(IN := FALSE);
				Internal.State 									:= USB_CONNECT_GET_LIST_CMD;
			ELSE
				Internal.CTON_Delay(IN := TRUE, PT := REAL_TO_TIME(delay*1000.0));
			END_IF;
 		USB_CONNECT_ERROR:
			connected 											:= FALSE;
	END_CASE;

	Internal.UsbNodeListGet_0();
	Internal.UsbNodeGet_0();
	Internal.DevLink_0();
	Internal.UsbMsDeviceReady_0();
	Internal.DevUnlink_0();

	IF connected THEN
		status													:= 0;
	END_IF;

END_FUNCTION_BLOCK
```

#### TC_Dir_Transfer.st
```iecst
(* Transfer List from Device to Another. Always Overwrites Existing. If either src or dest path includes directories, then the directories need to exist (this will not create them automatically) *)
FUNCTION_BLOCK TC_Dir_Transfer
	IF NOT enable THEN
		Internal.State 											:= TRANSFER_RESET;
	END_IF;

	CASE Internal.State OF
		TRANSFER_RESET:
			status												:= 65534;
			brsmemset(ADR(Internal),0,SIZEOF(Internal));
			Internal.State 										:= TRANSFER_IDLE;
		TRANSFER_IDLE:
			IF enable THEN
				IF pTransferList <> 0 THEN
					status										:= 65535;
					brsmemset(ADR(Internal),0,SIZEOF(Internal));
					Internal.ListIdx		 					:= 0;
					Internal.State 								:= TRANSFER_CHECK_LIST;
				ELSE
					status										:= 60001;
					Internal.State								:= TRANSFER_ERROR;
				END_IF;
			END_IF;
		TRANSFER_CHECK_LIST:
			status												:= 65535;
			IF Internal.ListIdx >= 0 AND Internal.ListIdx <= MAX_TRANSFER_LIST_IDX THEN
				brsmemcpy(ADR(Internal.TransferListItem),pTransferList+SIZEOF(Internal.TransferListItem)*Internal.ListIdx,SIZEOF(Internal.TransferListItem));
				IF Internal.TransferListItem.Valid THEN
					IF Internal.TransferListItem.SrcDelete AND Internal.TransferListItem.NoTransfer THEN
						IF Internal.TransferListItem.IsDir THEN
							Internal.State 						:= TRANSFER_DIR_DELETE_CMD;
						ELSE
							Internal.State 						:= TRANSFER_FILE_DELETE_CMD;
						END_IF;
					ELSIF Internal.TransferListItem.SrcCreateDir THEN
						Internal.State 							:= TRANSFER_DIR_CREATE_CMD;
					ELSIF Internal.TransferListItem.IsDir THEN
						Internal.State 							:= TRANSFER_DIR_COPY_CMD;
					ELSE
						Internal.State 							:= TRANSFER_FILE_COPY_CMD;
					END_IF;
				ELSE
					Internal.State 								:= TRANSFER_DONE;
				END_IF;
			ELSE
				Internal.State 									:= TRANSFER_DONE;
			END_IF;
		TRANSFER_DIR_COPY_CMD:
			status												:= 65535;
			Internal.DirCopy_0.enable 							:= TRUE;
			Internal.DirCopy_0.option 							:= fiOVERWRITE;
			Internal.DirCopy_0.pSrcDev 							:= ADR(Internal.TransferListItem.SrcDev);
			Internal.DirCopy_0.pSrcDir 							:= ADR(Internal.TransferListItem.SrcPath);
			Internal.DirCopy_0.pDestDev 						:= ADR(Internal.TransferListItem.DestDev);
			Internal.DirCopy_0.pDestDir 						:= ADR(Internal.TransferListItem.DestPath);
			Internal.State 										:= TRANSFER_DIR_COPY_WAIT;
		TRANSFER_DIR_COPY_WAIT:
			status												:= 65535;
			IF Internal.TransferListItem.SrcOrDestUSB AND NOT USB_Connected THEN
				Internal.DirCopy_0.enable 						:= FALSE;
				status											:= 65000;
				Internal.State 									:= TRANSFER_ERROR;
			ELSIF Internal.DirCopy_0.status = 0 THEN
				Internal.DirCopy_0.enable 						:= FALSE;
				IF Internal.TransferListItem.SrcDelete THEN
					Internal.State 								:= TRANSFER_DIR_DELETE_CMD;
				ELSE
					Internal.ListIdx							:= Internal.ListIdx + 1;
					Internal.State 								:= TRANSFER_CHECK_LIST;
				END_IF;
			ELSIF Internal.DirCopy_0.status <> ERR_FUB_BUSY AND Internal.DirCopy_0.status <> ERR_FUB_ENABLE_FALSE THEN
				Internal.DirCopy_0.enable 						:= FALSE;
				status											:= Internal.DirCopy_0.status;
				Internal.State 									:= TRANSFER_ERROR;
			END_IF;
		TRANSFER_DIR_DELETE_CMD:
			status												:= 65535;
			Internal.DirDeleteEx_0.enable 						:= TRUE;
			Internal.DirDeleteEx_0.pDevice 						:= ADR(Internal.TransferListItem.SrcDev);
			Internal.DirDeleteEx_0.pName	 					:= ADR(Internal.TransferListItem.SrcPath);
			Internal.State 										:= TRANSFER_DIR_DELETE_WAIT;
		TRANSFER_DIR_DELETE_WAIT:
			status												:= 65535;
			IF Internal.TransferListItem.SrcOrDestUSB AND NOT USB_Connected THEN
				Internal.DirDeleteEx_0.enable 					:= FALSE;
				status											:= 65000;
				Internal.State 									:= TRANSFER_ERROR;
			ELSIF Internal.DirDeleteEx_0.status = 0 THEN
				Internal.DirDeleteEx_0.enable 					:= FALSE;
				Internal.ListIdx								:= Internal.ListIdx + 1;
				Internal.State 									:= TRANSFER_CHECK_LIST;
			ELSIF Internal.DirDeleteEx_0.status <> ERR_FUB_BUSY AND Internal.DirDeleteEx_0.status <> ERR_FUB_ENABLE_FALSE THEN
				Internal.DirDeleteEx_0.enable 					:= FALSE;
				status											:= Internal.DirDeleteEx_0.status;
				Internal.State 									:= TRANSFER_ERROR;
			END_IF;
		TRANSFER_FILE_COPY_CMD:
			status												:= 65535;
			Internal.FileCopy_0.enable 							:= TRUE;
			Internal.FileCopy_0.option 							:= fiOVERWRITE;
			Internal.FileCopy_0.pSrcDev 						:= ADR(Internal.TransferListItem.SrcDev);
			Internal.FileCopy_0.pSrc	 						:= ADR(Internal.TransferListItem.SrcPath);
			Internal.FileCopy_0.pDestDev 						:= ADR(Internal.TransferListItem.DestDev);
			Internal.FileCopy_0.pDest							:= ADR(Internal.TransferListItem.DestPath);
			Internal.State 										:= TRANSFER_FILE_COPY_WAIT;
		TRANSFER_FILE_COPY_WAIT:
			status												:= 65535;
			IF Internal.TransferListItem.SrcOrDestUSB AND NOT USB_Connected THEN
				Internal.FileCopy_0.enable 						:= FALSE;
				status											:= 65000;
				Internal.State 									:= TRANSFER_ERROR;
			ELSIF Internal.FileCopy_0.status = 0 THEN
				Internal.FileCopy_0.enable 						:= FALSE;
				IF Internal.TransferListItem.SrcDelete THEN
					Internal.State 								:= TRANSFER_FILE_DELETE_CMD;
				ELSE
					Internal.ListIdx							:= Internal.ListIdx + 1;
					Internal.State 								:= TRANSFER_CHECK_LIST;
				END_IF;
			ELSIF Internal.FileCopy_0.status <> ERR_FUB_BUSY AND Internal.FileCopy_0.status <> ERR_FUB_ENABLE_FALSE THEN
				Internal.FileCopy_0.enable 						:= FALSE;
				status											:= Internal.FileCopy_0.status;
				Internal.State 									:= TRANSFER_ERROR;
			END_IF;
		TRANSFER_FILE_DELETE_CMD:
			status												:= 65535;
			Internal.FileDelete_0.enable 						:= TRUE;
			Internal.FileDelete_0.pDevice 						:= ADR(Internal.TransferListItem.SrcDev);
			Internal.FileDelete_0.pName	 						:= ADR(Internal.TransferListItem.SrcPath);
			Internal.State 										:= TRANSFER_FILE_DELETE_WAIT;
		TRANSFER_FILE_DELETE_WAIT:
			status												:= 65535;
			IF Internal.TransferListItem.SrcOrDestUSB AND NOT USB_Connected THEN
				Internal.FileDelete_0.enable 					:= FALSE;
				status											:= 65000;
				Internal.State 									:= TRANSFER_ERROR;
			ELSIF Internal.FileDelete_0.status = 0 THEN
				Internal.FileDelete_0.enable 					:= FALSE;
				Internal.ListIdx								:= Internal.ListIdx + 1;
				Internal.State 									:= TRANSFER_CHECK_LIST;
			ELSIF Internal.FileDelete_0.status <> ERR_FUB_BUSY AND Internal.FileDelete_0.status <> ERR_FUB_ENABLE_FALSE THEN
				Internal.FileDelete_0.enable 					:= FALSE;
				status											:= Internal.FileDelete_0.status;
				Internal.State 									:= TRANSFER_ERROR;
			END_IF;
		TRANSFER_DIR_CREATE_CMD:
			status												:= 65535;
			Internal.DirCreate_0.enable 						:= TRUE;
			Internal.DirCreate_0.pDevice 						:= ADR(Internal.TransferListItem.SrcDev);
			Internal.DirCreate_0.pName	 						:= ADR(Internal.TransferListItem.SrcPath);
			Internal.State 										:= TRANSFER_DIR_CREATE_WAIT;
		TRANSFER_DIR_CREATE_WAIT:
			status												:= 65535;
			IF Internal.TransferListItem.SrcOrDestUSB AND NOT USB_Connected THEN
				Internal.DirCreate_0.enable 					:= FALSE;
				status											:= 65000;
				Internal.State 									:= TRANSFER_ERROR;
			ELSIF Internal.DirCreate_0.status = 0 THEN
				Internal.DirCreate_0.enable 					:= FALSE;
				Internal.ListIdx								:= Internal.ListIdx + 1;
				Internal.State 									:= TRANSFER_CHECK_LIST;
			ELSIF Internal.DirCreate_0.status <> ERR_FUB_BUSY AND Internal.DirCreate_0.status <> ERR_FUB_ENABLE_FALSE THEN
				Internal.FileDelete_0.enable 					:= FALSE;
				status											:= Internal.DirCreate_0.status;
				Internal.State 									:= TRANSFER_ERROR;
			END_IF;
		TRANSFER_DONE:
			status												:= 0;
		TRANSFER_ERROR:
			// Error
	END_CASE;

	index 														:= Internal.ListIdx;

	Internal.DirCreate_0();
	Internal.DirCopy_0();
	Internal.FileCopy_0();
	Internal.DirDeleteEx_0();
	Internal.FileDelete_0();

END_FUNCTION_BLOCK
```

#### TC_DirReadAll.st
```iecst
(* Reads Entire File Device *)
FUNCTION_BLOCK TC_DirReadAll
	IF enable = FALSE THEN
		Internal.State														:= DIRREADALL_RESET;
	END_IF;

	CASE Internal.State OF
		DIRREADALL_RESET:
			status															:= 65534;
			brsmemset(ADR(Internal),0,SIZEOF(Internal));
			Internal.State													:= DIRREADALL_IDLE;
		DIRREADALL_IDLE:
			status															:= 65534;
			IF enable THEN
				IF pDevice <> 0 AND pFileList <> 0 THEN
					brsmemset(ADR(Internal),0,SIZEOF(Internal));
					brsmemset(pFileList,0,(SIZEOF(Internal.FileListItem)*(MAX_DIR_MAN_FILE_LIST_IDX+1)));
					Internal.FileListItem.DateUDINT := 0;
					Internal.FileListItem.IsDir := TRUE;
					Internal.FileListItem.Path := '';
					Internal.FileListItem.Size := 0;
					Internal.FileListItem.Internal.0 := 0;
					Internal.FileListIdx									:= 0;
					IF Internal.FileListIdx <= MAX_DIR_MAN_FILE_LIST_IDX THEN
						brsmemcpy(pFileList+SIZEOF(Internal.FileListItem)*Internal.FileListIdx,ADR(Internal.FileListItem),SIZEOF(Internal.FileListItem));
					END_IF;
					Internal.FileListIdx									:= Internal.FileListIdx + 1;
					status													:= 65535;
					Internal.CurrentDirPath									:= '';
					Internal.State											:= DIRREADALL_OPEN_CMD;
				ELSE
					brsmemset(ADR(Internal),0,SIZEOF(Internal));
					status													:= 60001;
					Internal.State											:= DIRREADALL_ERROR;
				END_IF;
			END_IF;
		DIRREADALL_OPEN_CMD:
			status															:= 65535;
			Internal.DirOpen_0.enable 										:= TRUE;
			Internal.DirOpen_0.pDevice 										:= pDevice;
			Internal.DirOpen_0.pName 										:= ADR(Internal.CurrentDirPath);
			Internal.State 													:= DIRREADALL_OPEN_WAIT;
		DIRREADALL_OPEN_WAIT:
			status															:= 65535;
			IF Internal.DirOpen_0.status = 0 THEN
				Internal.DirOpen_0.enable 									:= FALSE;
				Internal.DirIdent 											:= Internal.DirOpen_0.ident;
				Internal.State 												:= DIRREADALL_READ_CMD;
			ELSIF Internal.DirOpen_0.status <> ERR_FUB_BUSY AND Internal.DirOpen_0.status <> ERR_FUB_ENABLE_FALSE THEN
				Internal.DirOpen_0.enable 									:= FALSE;
				status														:= Internal.DirOpen_0.status;
				Internal.State 												:= DIRREADALL_ERROR;
			END_IF;
		DIRREADALL_READ_CMD:
			status															:= 65535;
			brsmemset(ADR(Internal.DirData),0,SIZEOF(Internal.DirData));
			Internal.DirReadEx_0.enable 									:= TRUE;
			Internal.DirReadEx_0.ident 										:= Internal.DirIdent;
			Internal.DirReadEx_0.pData 										:= ADR(Internal.DirData);
			Internal.DirReadEx_0.data_len 									:= SIZEOF(Internal.DirData);
			Internal.State 													:= DIRREADALL_READ_WAIT;
		DIRREADALL_READ_WAIT:
			status															:= 65535;
			IF Internal.DirReadEx_0.status = 0 THEN
				Internal.DirReadEx_0.enable 								:= FALSE;
				brsmemset(ADR(Internal.FileListItem),0,SIZEOF(Internal.FileListItem));
				IF Internal.DirData.Filename[0] <> 46 THEN // check for '.' or '..' and filter out, '.' is decimal 46 in ascii
					IF Internal.CurrentDirPath <> '' THEN
						brsstrcat(ADR(Internal.FileListItem.Path),ADR(Internal.CurrentDirPath));
						brsstrcat(ADR(Internal.FileListItem.Path),ADR('/'));
					END_IF;
					brsstrcat(ADR(Internal.FileListItem.Path),ADR(Internal.DirData.Filename));
					Internal.FileListItem.DateUDINT 						:= DT_TO_UDINT(Internal.DirData.Date);
					Internal.FileListItem.Size 								:= Internal.DirData.Filelength;
					Internal.FileListItem.IsDir 							:= Internal.DirData.Mode = 1;
					Internal.FileListItem.Internal.0						:= Internal.DirData.Mode = 1;
					IF Internal.FileListIdx >= MAX_DIR_MAN_FILE_LIST_IDX THEN
						Internal.State 										:= DIRREADALL_CLOSE_WAIT;
						Internal.DirClose_0.ident 							:= Internal.DirIdent;
						Internal.DirClose_0.enable 							:= TRUE;
					ELSE
						brsmemcpy(pFileList+SIZEOF(Internal.FileListItem)*Internal.FileListIdx,ADR(Internal.FileListItem),SIZEOF(Internal.FileListItem));
						Internal.FileListIdx								:= Internal.FileListIdx + 1;
						Internal.State 										:= DIRREADALL_READ_CMD;
					END_IF;
				ELSE
					Internal.State 											:= DIRREADALL_READ_CMD;
				END_IF;
			ELSIF Internal.DirReadEx_0.status <> ERR_FUB_BUSY AND Internal.DirReadEx_0.status <> ERR_FUB_ENABLE_FALSE THEN
				Internal.DirReadEx_0.enable 								:= FALSE;
				Internal.DirClose_0.ident 									:= Internal.DirIdent;
				Internal.DirClose_0.enable 									:= TRUE;
				Internal.State 												:= DIRREADALL_CLOSE_WAIT;
			END_IF;
		DIRREADALL_CLOSE_WAIT:
			status															:= 65535;
			IF Internal.DirClose_0.status = 0 OR (Internal.DirClose_0.status <> ERR_FUB_BUSY AND Internal.DirClose_0.status <> ERR_FUB_ENABLE_FALSE) THEN
				Internal.DirClose_0.enable 									:= FALSE;
				IF Internal.FileListIdx >= MAX_DIR_MAN_FILE_LIST_IDX THEN
					Internal.State 											:= DIRREADALL_EVALUATE;
				ELSE
					FOR Internal.i := 0 TO MAX_DIR_MAN_FILE_LIST_IDX DO
						brsmemcpy(ADR(Internal.FileListItem),pFileList+SIZEOF(Internal.FileListItem)*Internal.i,SIZEOF(Internal.FileListItem));
						IF Internal.FileListItem.Path = '' AND Internal.FileListItem.IsDir = FALSE THEN
							Internal.State 									:= DIRREADALL_EVALUATE;
							EXIT;
						ELSIF Internal.FileListItem.Internal.0 = 1 THEN
							Internal.CurrentDirPath							:= Internal.FileListItem.Path;
							Internal.FileListItem.Internal.0				:= 0;
							brsmemcpy(pFileList+SIZEOF(Internal.FileListItem)*Internal.i,ADR(Internal.FileListItem),SIZEOF(Internal.FileListItem));
							Internal.State 									:= DIRREADALL_OPEN_CMD;
							EXIT;
						END_IF;
					END_FOR;
				END_IF;
			END_IF;
		DIRREADALL_EVALUATE:
			status															:= 65535;
//			// Build Lists
//			FOR Internal.i := 0 TO MAX_DIR_MAN_FILE_LIST_IDX DO
//				IF Internal.FileList[Internal.i].Path = '' THEN
//					EXIT;
//				ELSIF Internal.FileList[Internal.i].IsDir THEN
//					FileList[Internal.FileListIdx] 							:= Internal.FileList[Internal.i];
//					IF Internal.FileListIdx < MAX_DIR_MAN_FILE_LIST_IDX THEN
//						Internal.FileListIdx								:= Internal.FileListIdx + 1;
//					END_IF;
//				ELSE
//					FileList[Internal.FileListIdx] 							:= Internal.FileList[Internal.i];
//					IF Internal.FileListIdx < MAX_DIR_MAN_FILE_LIST_IDX THEN
//						Internal.FileListIdx								:= Internal.FileListIdx + 1;
//					END_IF;
//				END_IF;
//			END_FOR;
//			FileList 														:= Internal.FileList;
//			Internal.FileListIdx 											:= 0;
			Internal.State 													:= DIRREADALL_DONE;
		DIRREADALL_DONE:
			status															:= 0;
		DIRREADALL_ERROR:
			// Error
	END_CASE;

	Internal.DirOpen_0();
	Internal.DirReadEx_0();
	Internal.DirClose_0();

END_FUNCTION_BLOCK
```

### Library Logical/Libraries/TC_Convert (IEC)

#### Types.typ - Exported data types
```iecst
TYPE
	TC_DT_Parser_Internal_typ : 	STRUCT
		DateTime : DATE_AND_TIME;
		dateTimeStruct : DTStructure;
		year : STRING[4];
		month : STRING[2];
		day : STRING[2];
		hour : STRING[2];
		minute : STRING[2];
		second : STRING[2];
	END_STRUCT;
	TC_DT_Formatter_Internal_typ : 	STRUCT
		dateTimeStruct : DTStructure;
		year : STRING[4];
		month : STRING[2];
		day : STRING[2];
		hour : STRING[2];
		minute : STRING[2];
		second : STRING[2];
		separator : STRING[1];
		c : USINT;
		i : UDINT;
		formatLen : UDINT;
		format : STRING[80];
		output : STRING[80];
		length : UDINT;
	END_STRUCT;
END_TYPE
```

#### TC_Convert.fun - Exported functions and function blocks
```iecst
FUNCTION TC_DT_Parser : BOOL
	VAR_INPUT
		pValueString : UDINT;
		pOutDT : UDINT;
	END_VAR
	VAR
		Internal : TC_DT_Parser_Internal_typ;
	END_VAR
END_FUNCTION

FUNCTION TC_DT_Formatter : BOOL
	VAR_INPUT
		value : DATE_AND_TIME;
		pInFormatString : UDINT; (*Optional*)
		pOutString : UDINT;
		OutStringLength : UDINT;
	END_VAR
	VAR
		Internal : TC_DT_Formatter_Internal_typ;
	END_VAR
END_FUNCTION
```

#### TC_DT_Formatter.st
```iecst
(* Formats DATE_AND_TIME Value into a string *)
FUNCTION TC_DT_Formatter
	TC_DT_Formatter 								:= TRUE;
	IF pOutString = 0 OR OutStringLength = 0 THEN
		TC_DT_Formatter 							:= FALSE;
	ELSE
		TC_DT_Formatter 							:= TRUE;
		Internal.output								:= '';
		Internal.formatLen 							:= brsstrlen(pInFormatString);
		IF pInFormatString = 0 OR Internal.formatLen = 0 OR Internal.formatLen > SIZEOF(Internal.format)-1 THEN
			Internal.format 						:= 'DT#y-m-d-h:M:s';
			Internal.formatLen 						:= brsstrlen(ADR(Internal.format));
		ELSE
			brsstrcpy(ADR(Internal.format),pInFormatString);
			Internal.formatLen 						:= brsstrlen(ADR(Internal.format));
		END_IF;
		DT_TO_DTStructure(value,ADR(Internal.dateTimeStruct));
		Internal.year 								:= UINT_TO_STRING(Internal.dateTimeStruct.year);
		Internal.month 								:= USINT_TO_STRING(Internal.dateTimeStruct.month);
		Internal.day 								:= USINT_TO_STRING(Internal.dateTimeStruct.day);
		Internal.hour 								:= USINT_TO_STRING(Internal.dateTimeStruct.hour);
		Internal.minute 							:= USINT_TO_STRING(Internal.dateTimeStruct.minute);
		Internal.second 							:= USINT_TO_STRING(Internal.dateTimeStruct.second);
		FOR Internal.i := 0 TO Internal.formatLen DO
			brsmemcpy(ADR(Internal.c),ADR(Internal.format)+Internal.i,1);
		    CASE Internal.c OF
		        121: //'y'
					IF Internal.length + 4 >= OutStringLength-1 THEN
						Internal.output 			:= '';
						TC_DT_Formatter 			:= FALSE;
						RETURN;
					ELSE
						Internal.length				:= brsstrcat(ADR(Internal.output),ADR(Internal.year)) - ADR(Internal.output);
					END_IF;
		        109: //'m'
					IF Internal.length + 2 >= OutStringLength-1 THEN
						Internal.output 			:= '';
						TC_DT_Formatter 			:= FALSE;
						RETURN;
					ELSE
						IF Internal.dateTimeStruct.month <= 9 THEN
							brsstrcat(ADR(Internal.output),ADR('0'));
						END_IF;
						Internal.length				:= brsstrcat(ADR(Internal.output),ADR(Internal.month)) - ADR(Internal.output);
					END_IF;
		        100: //'d'
					IF Internal.length + 2 >= OutStringLength-1 THEN
						Internal.output 			:= '';
						TC_DT_Formatter 			:= FALSE;
						RETURN;
					ELSE
						IF Internal.dateTimeStruct.day <= 9 THEN
							brsstrcat(ADR(Internal.output),ADR('0'));
						END_IF;
						Internal.length				:= brsstrcat(ADR(Internal.output),ADR(Internal.day)) - ADR(Internal.output);
					END_IF;
		        104: //'h'
					IF Internal.length + 2 >= OutStringLength-1 THEN
						Internal.output 			:= '';
						TC_DT_Formatter 			:= FALSE;
						RETURN;
					ELSE
						IF Internal.dateTimeStruct.hour <= 9 THEN
							brsstrcat(ADR(Internal.output),ADR('0'));
						END_IF;
						Internal.length				:= brsstrcat(ADR(Internal.output),ADR(Internal.hour)) - ADR(Internal.output);
					END_IF;
		        77: //'M'
					IF Internal.length + 2 >= OutStringLength-1 THEN
						Internal.output 			:= '';
						TC_DT_Formatter 			:= FALSE;
						RETURN;
					ELSE
						IF Internal.dateTimeStruct.minute <= 9 THEN
							brsstrcat(ADR(Internal.output),ADR('0'));
						END_IF;
						Internal.length				:= brsstrcat(ADR(Internal.output),ADR(Internal.minute)) - ADR(Internal.output);
					END_IF;
		        115: //'s'
					IF Internal.length + 2 >= OutStringLength-1 THEN
						Internal.output 			:= '';
						TC_DT_Formatter 			:= FALSE;
						RETURN;
					ELSE
						IF Internal.dateTimeStruct.second <= 9 THEN
							brsstrcat(ADR(Internal.output),ADR('0'));
						END_IF;
						Internal.length				:= brsstrcat(ADR(Internal.output),ADR(Internal.second)) - ADR(Internal.output);
					END_IF;
		        ELSE
					brsmemset(ADR(Internal.separator),0,SIZEOF(Internal.separator));
					brsmemcpy(ADR(Internal.separator),ADR(Internal.c),1);
					IF Internal.length + 1 >= OutStringLength-1 THEN
						Internal.output 			:= '';
						TC_DT_Formatter 			:= FALSE;
						RETURN;
					ELSE
						Internal.length				:= brsstrcat(ADR(Internal.output),ADR(Internal.separator)) - ADR(Internal.output);
					END_IF;
		    END_CASE
		END_FOR;
		IF NOT TC_DT_Formatter THEN
			brsmemset(pOutString,0,OutStringLength);
		ELSE
			brsstrcpy(pOutString,ADR(Internal.output));
		END_IF;
	END_IF;
END_FUNCTION
```

#### TC_DT_Parser.st
```iecst
(* Parses string into DATE_AND_TIME format !!!!!STRING MUST BE IN THE FORM OF DT#yyyy-mm-dd-hh:MM:ss!!!!! all other will fail*)
FUNCTION TC_DT_Parser
	TC_DT_Parser 						:= TRUE;
	IF pOutDT = 0 OR pValueString = 0 THEN
		TC_DT_Parser 					:= FALSE;
	ELSE
		TC_DT_Parser					:= TRUE;
		brsmemset(ADR(Internal),0,SIZEOF(Internal));
		brsmemcpy(ADR(Internal.year),pValueString+3,4);
		brsmemcpy(ADR(Internal.month),pValueString+8,2);
		brsmemcpy(ADR(Internal.day),pValueString+11,2);
		brsmemcpy(ADR(Internal.hour),pValueString+14,2);
		brsmemcpy(ADR(Internal.minute),pValueString+17,2);
		brsmemcpy(ADR(Internal.second),pValueString+20,2);
		Internal.dateTimeStruct.year	:= STRING_TO_UINT(Internal.year);
		Internal.dateTimeStruct.month	:= STRING_TO_USINT(Internal.month);
		Internal.dateTimeStruct.day		:= STRING_TO_USINT(Internal.day);
		Internal.dateTimeStruct.hour	:= STRING_TO_USINT(Internal.hour);
		Internal.dateTimeStruct.minute	:= STRING_TO_USINT(Internal.minute);
		Internal.dateTimeStruct.second	:= STRING_TO_USINT(Internal.second);
		Internal.DateTime := DTStructure_TO_DT(ADR(Internal.dateTimeStruct));
		brsmemcpy(pOutDT,ADR(Internal.DateTime),SIZEOF(Internal.DateTime));
	END_IF;
END_FUNCTION
```

### Library Logical/Libraries/TC_ItemX (IEC)

#### Types.typ - Exported data types
```iecst
TYPE
	ItemX_typ : 	STRUCT
		CurrentUID : UDINT; (*REQUIRED*)
		ValidIndex : BOOL; (*REQUIRED*)
		ReturnedIndex : INT; (*REQUIRED*)
		Elem : ItemX_Elem_typ; (*REQUIRED*)
		List : ARRAY[0..MAX_ITEM_X_IDX]OF ItemX_Elem_typ; (*REQUIRED*)
	END_STRUCT;
	ItemX_Elem_typ : 	STRUCT
		UID : UDINT; (*REQUIRED*)
		State : ITEM_X_STATE_ENUM; (*REQUIRED*)
		LastLoc : ITEM_X_LOC_ENUM; (*REQUIRED*)
		Loc : ITEM_X_LOC_ENUM; (*REQUIRED*)
		Par : ItemX_Par_typ; (*REQUIRED*)
		Status : ItemX_Status_typ; (*REQUIRED*)
	END_STRUCT;
	ItemX_Status_typ : 	STRUCT
		Position : REAL;
		Length : REAL;
		ManuallyRemoved : BOOL;
		Rejected : BOOL;
		Passed : BOOL;
		TimeIn : DATE_AND_TIME;
		TimeOut : DATE_AND_TIME;
		Error : BOOL;
	END_STRUCT;
	ItemX_Par_typ : 	STRUCT
		ProductID : INT;
		Recipe : ItemX_Par_Recipe_typ;
	END_STRUCT;
	ItemX_Par_Recipe_typ : 	STRUCT
		MaxLength : REAL;
	END_STRUCT;
	ITEM_X_STATE_ENUM :
		(
		ITEM_X_STATE_UNDEFINED, (*REQUIRED*)
		ITEM_X_STATE_WAIT_START,
		ITEM_X_STATE_ACTIVE,
		ITEM_X_STATE_DONE,
		ITEM_X_STATE_UNKNOWN,
		ITEM_X_STATE_ERRORSTOP
		);
	ITEM_X_LOC_ENUM :
		(
		ITEM_X_LOC_UNDEFINED, (*REQUIRED*)
		ITEM_X_LOC_UNKNOWN
		);
	TC_ItemX_Internal_typ : 	STRUCT
		i : INT;
		j : INT;
		tempItemX : ItemX_Elem_typ;
		tempIndex : INT;
		tempUID : UDINT;
	END_STRUCT;
END_TYPE
```

#### TC_ItemX.fun - Exported functions and function blocks
```iecst
{REDUND_ERROR} FUNCTION TC_ItemX_DeleteByIndex : BOOL (* *) (*$GROUP=User,$CAT=User,$GROUPICON=User.png,$CATICON=User.png*)
	VAR_INPUT
		Index : INT;
	END_VAR
	VAR_IN_OUT
		ItemX : ItemX_typ;
	END_VAR
	VAR
		Internal : TC_ItemX_Internal_typ;
	END_VAR
END_FUNCTION

{REDUND_ERROR} FUNCTION TC_ItemX_DeleteByUID : BOOL (* *) (*$GROUP=User,$CAT=User,$GROUPICON=User.png,$CATICON=User.png*)
	VAR_INPUT
		UID : UDINT;
	END_VAR
	VAR_IN_OUT
		ItemX : ItemX_typ;
	END_VAR
	VAR
		Internal : TC_ItemX_Internal_typ;
	END_VAR
END_FUNCTION

{REDUND_ERROR} FUNCTION TC_ItemX_UID_TO_Index : BOOL (* *) (*$GROUP=User,$CAT=User,$GROUPICON=User.png,$CATICON=User.png*)
	VAR_INPUT
		UID : UDINT;
	END_VAR
	VAR_IN_OUT
		ItemX : ItemX_typ;
	END_VAR
	VAR
		Internal : TC_ItemX_Internal_typ;
	END_VAR
END_FUNCTION

{REDUND_ERROR} FUNCTION TC_ItemX_Sanitize : BOOL (* *) (*$GROUP=User,$CAT=User,$GROUPICON=User.png,$CATICON=User.png*)
	VAR_IN_OUT
		ItemX : ItemX_typ;
	END_VAR
	VAR
		Internal : TC_ItemX_Internal_typ;
	END_VAR
END_FUNCTION

{REDUND_ERROR} FUNCTION TC_ItemX_Reorder_LowToHighUID : BOOL (* *) (*$GROUP=User,$CAT=User,$GROUPICON=User.png,$CATICON=User.png*)
	VAR_IN_OUT
		ItemX : ItemX_typ;
	END_VAR
	VAR
		Internal : TC_ItemX_Internal_typ;
	END_VAR
END_FUNCTION

{REDUND_ERROR} FUNCTION TC_ItemX_Reorder_HighToLowUID : BOOL (* *) (*$GROUP=User,$CAT=User,$GROUPICON=User.png,$CATICON=User.png*)
	VAR_IN_OUT
		ItemX : ItemX_typ;
	END_VAR
	VAR
		Internal : TC_ItemX_Internal_typ;
	END_VAR
END_FUNCTION

{REDUND_ERROR} FUNCTION TC_ItemX_IndexLowestUID : BOOL (* *) (*$GROUP=User,$CAT=User,$GROUPICON=User.png,$CATICON=User.png*)
	VAR_IN_OUT
		ItemX : ItemX_typ;
	END_VAR
	VAR
		Internal : TC_ItemX_Internal_typ;
	END_VAR
END_FUNCTION

{REDUND_ERROR} FUNCTION TC_ItemX_IndexHighestUID : BOOL (* *) (*$GROUP=User,$CAT=User,$GROUPICON=User.png,$CATICON=User.png*)
	VAR_IN_OUT
		ItemX : ItemX_typ;
	END_VAR
	VAR
		Internal : TC_ItemX_Internal_typ;
	END_VAR
END_FUNCTION

{REDUND_ERROR} FUNCTION TC_ItemX_FirstOpenIndex : BOOL (* *) (*$GROUP=User,$CAT=User,$GROUPICON=User.png,$CATICON=User.png*)
	VAR_IN_OUT
		ItemX : ItemX_typ;
	END_VAR
	VAR
		Internal : TC_ItemX_Internal_typ;
	END_VAR
END_FUNCTION

{REDUND_ERROR} FUNCTION TC_ItemX_GetElemByIndex : BOOL (* *) (*$GROUP=User,$CAT=User,$GROUPICON=User.png,$CATICON=User.png*)
	VAR_INPUT
		Index : INT;
	END_VAR
	VAR_IN_OUT
		ItemX : ItemX_typ;
	END_VAR
	VAR
		Internal : TC_ItemX_Internal_typ;
	END_VAR
END_FUNCTION

{REDUND_ERROR} FUNCTION TC_ItemX_GetElemByUID : BOOL (* *) (*$GROUP=User,$CAT=User,$GROUPICON=User.png,$CATICON=User.png*)
	VAR_INPUT
		UID : UDINT;
	END_VAR
	VAR_IN_OUT
		ItemX : ItemX_typ;
	END_VAR
	VAR
		Internal : TC_ItemX_Internal_typ;
	END_VAR
END_FUNCTION

{REDUND_ERROR} FUNCTION TC_ItemX_ModElemByIndex : BOOL (* *) (*$GROUP=User,$CAT=User,$GROUPICON=User.png,$CATICON=User.png*)
	VAR_INPUT
		Index : INT;
	END_VAR
	VAR_IN_OUT
		ItemX : ItemX_typ;
	END_VAR
	VAR
		Internal : TC_ItemX_Internal_typ;
	END_VAR
END_FUNCTION

{REDUND_ERROR} FUNCTION TC_ItemX_ModElemByUID : BOOL (* *) (*$GROUP=User,$CAT=User,$GROUPICON=User.png,$CATICON=User.png*)
	VAR_INPUT
		UID : UDINT;
	END_VAR
	VAR_IN_OUT
		ItemX : ItemX_typ;
	END_VAR
	VAR
		Internal : TC_ItemX_Internal_typ;
	END_VAR
END_FUNCTION

{REDUND_ERROR} FUNCTION TC_ItemX_AddElem : BOOL (* *) (*$GROUP=User,$CAT=User,$GROUPICON=User.png,$CATICON=User.png*)
	VAR_IN_OUT
		ItemX : ItemX_typ;
	END_VAR
	VAR
		Internal : TC_ItemX_Internal_typ;
	END_VAR
END_FUNCTION

{REDUND_ERROR} FUNCTION TC_ItemX_IncrementUID : BOOL (* *) (*$GROUP=User,$CAT=User,$GROUPICON=User.png,$CATICON=User.png*)
	VAR_IN_OUT
		ItemX : ItemX_typ;
	END_VAR
	VAR
		Internal : TC_ItemX_Internal_typ;
	END_VAR
END_FUNCTION
```

#### TC_ItemX_FirstOpenIndex.st
```iecst
(* Finds the first open index of the item array *)
FUNCTION TC_ItemX_FirstOpenIndex
	TC_ItemX_FirstOpenIndex							:= FALSE;
	ItemX.ReturnedIndex								:= -1;
	FOR Internal.i := 0 TO MAX_ITEM_X_IDX DO
		IF ItemX.List[Internal.i].UID = 0 THEN
			TC_ItemX_FirstOpenIndex					:= TRUE;
			ItemX.ReturnedIndex						:= Internal.i;
			EXIT;
		END_IF;
	END_FOR;

	// This is here for keeping the ItemX structure up to date and should be at the bottom of every function call in the library
	ItemX.ValidIndex									:= FALSE;
	IF ItemX.ReturnedIndex >= 0 AND ItemX.ReturnedIndex <= MAX_ITEM_X_IDX THEN
		ItemX.ValidIndex								:= TRUE;
	END_IF;

END_FUNCTION
```

#### TC_ItemX_UID_TO_Index.st
```iecst
(* Returns the first index matching the UID entered *)
FUNCTION TC_ItemX_UID_TO_Index
	TC_ItemX_UID_TO_Index							:= FALSE;
	ItemX.ReturnedIndex								:= -1;
	FOR Internal.i := 0 TO MAX_ITEM_X_IDX DO
		IF ItemX.List[Internal.i].UID = UID THEN
			TC_ItemX_UID_TO_Index					:= TRUE;
			ItemX.ReturnedIndex						:= Internal.i;
			EXIT;
		END_IF;
	END_FOR;

	// This is here for keeping the ItemX structure up to date and should be at the bottom of every function call in the library
	ItemX.ValidIndex									:= FALSE;
	IF ItemX.ReturnedIndex >= 0 AND ItemX.ReturnedIndex <= MAX_ITEM_X_IDX THEN
		ItemX.ValidIndex								:= TRUE;
	END_IF;

END_FUNCTION
```

#### TC_ItemX_DeleteByUID.st
```iecst
(* Deletes the first index matching the UID entered, Returns True if Deleted, False if not found *)
FUNCTION TC_ItemX_DeleteByUID
	TC_ItemX_DeleteByUID								:= FALSE;
	ItemX.ReturnedIndex								:= -1;
	FOR Internal.i := 0 TO MAX_ITEM_X_IDX DO
		IF ItemX.List[Internal.i].UID = UID THEN
			brsmemset(ADR(ItemX.List[Internal.i]),0,SIZEOF(ItemX.List[Internal.i]));
			ItemX.ReturnedIndex						:= Internal.i;
			TC_ItemX_DeleteByUID						:= TRUE;
			EXIT;
		END_IF;
	END_FOR;

	// This is here for keeping the ItemX structure up to date and should be at the bottom of every function call in the library
	ItemX.ValidIndex									:= FALSE;
	IF ItemX.ReturnedIndex >= 0 AND ItemX.ReturnedIndex <= MAX_ITEM_X_IDX THEN
		ItemX.ValidIndex								:= TRUE;
	END_IF;

END_FUNCTION
```

#### TC_ItemX_DeleteByIndex.st
```iecst
(* Deletes the index entered, Returns True if Deleted, False if not in range *)
FUNCTION TC_ItemX_DeleteByIndex
	Internal.i 											:= 0; // This is to avoid a compiler warning that internal is not used.
	TC_ItemX_DeleteByIndex								:= FALSE;
	ItemX.ReturnedIndex									:= -1;
	IF Index >= 0 AND Index <= MAX_ITEM_X_IDX THEN
		brsmemset(ADR(ItemX.List[Index]),0,SIZEOF(ItemX.List[Index]));
		ItemX.ReturnedIndex								:= Index;
		TC_ItemX_DeleteByIndex							:= TRUE;
	END_IF;

	// This is here for keeping the ItemX structure up to date and should be at the bottom of every function call in the library
	ItemX.ValidIndex									:= FALSE;
	IF ItemX.ReturnedIndex >= 0 AND ItemX.ReturnedIndex <= MAX_ITEM_X_IDX THEN
		ItemX.ValidIndex								:= TRUE;
	END_IF;

END_FUNCTION
```

#### TC_ItemX_IndexLowestUID.st
```iecst
(* Returns the index of the lowest UID found in the item array,*)
FUNCTION TC_ItemX_IndexLowestUID
	TC_ItemX_IndexLowestUID							:= FALSE;
	ItemX.ReturnedIndex								:= -1;
	Internal.tempUID								:= 4294967295; // Set to UDINT max
	FOR Internal.i := 0 TO MAX_ITEM_X_IDX DO
		IF ItemX.List[Internal.i].UID < Internal.tempUID AND ItemX.List[Internal.i].UID > 0 THEN
			Internal.tempUID						:= ItemX.List[Internal.i].UID;
			ItemX.ReturnedIndex						:= Internal.i;
			TC_ItemX_IndexLowestUID					:= TRUE;
		END_IF;
	END_FOR;

	// This is here for keeping the ItemX structure up to date and should be at the bottom of every function call in the library
	ItemX.ValidIndex									:= FALSE;
	IF ItemX.ReturnedIndex >= 0 AND ItemX.ReturnedIndex <= MAX_ITEM_X_IDX THEN
		ItemX.ValidIndex								:= TRUE;
	END_IF;

END_FUNCTION
```

#### TC_ItemX_IndexHighestUID.st
```iecst
(* Returns the index of the highest UID found in the item array, -1 if All UID are 0 *)
FUNCTION TC_ItemX_IndexHighestUID
	TC_ItemX_IndexHighestUID							:= FALSE;
	ItemX.ReturnedIndex								:= -1;
	Internal.tempUID								:= 0;
	FOR Internal.i := 0 TO MAX_ITEM_X_IDX DO
		IF ItemX.List[Internal.i].UID > Internal.tempUID THEN
			Internal.tempUID						:= ItemX.List[Internal.i].UID;
			ItemX.ReturnedIndex						:= Internal.i;
			TC_ItemX_IndexHighestUID					:= TRUE;
		END_IF;
	END_FOR;

	// This is here for keeping the ItemX structure up to date and should be at the bottom of every function call in the library
	ItemX.ValidIndex									:= FALSE;
	IF ItemX.ReturnedIndex >= 0 AND ItemX.ReturnedIndex <= MAX_ITEM_X_IDX THEN
		ItemX.ValidIndex								:= TRUE;
	END_IF;

END_FUNCTION
```

#### TC_ItemX_Reorder_HighToLowUID.st
```iecst
(* Reorders the array to be from high to low in terms of UID *)
FUNCTION TC_ItemX_Reorder_HighToLowUID
	TC_ItemX_Reorder_HighToLowUID					:= TRUE;
	FOR Internal.i := 0 TO MAX_ITEM_X_IDX DO
		// Find Next Highest Index
		Internal.tempIndex							:= Internal.i;
		FOR Internal.j := Internal.i TO MAX_ITEM_X_IDX DO
			IF ItemX.List[Internal.j].UID > ItemX.List[Internal.tempIndex].UID THEN
				Internal.tempIndex					:= Internal.j;
			END_IF;
		END_FOR;
		// Swap ItemXs
		Internal.tempItemX							:= ItemX.List[Internal.i];
		ItemX.List[Internal.i]						:= ItemX.List[Internal.tempIndex];
		ItemX.List[Internal.tempIndex]				:= Internal.tempItemX;
		IF ItemX.List[Internal.i].UID = 0 THEN
			ItemX.ReturnedIndex 						:= Internal.i;
			EXIT;
		END_IF;
	END_FOR;

	// This is here for keeping the ItemX structure up to date and should be at the bottom of every function call in the library
	ItemX.ValidIndex									:= FALSE;
	IF ItemX.ReturnedIndex >= 0 AND ItemX.ReturnedIndex <= MAX_ITEM_X_IDX THEN
		ItemX.ValidIndex								:= TRUE;
	END_IF;

END_FUNCTION
```

#### TC_ItemX_Reorder_LowToHighUID.st
```iecst
(* Reorders the array to be from low to high in terms of UID, 0 elements left at the end of the array *)
FUNCTION TC_ItemX_Reorder_LowToHighUID
	TC_ItemX_Reorder_LowToHighUID					:= TRUE;
	FOR Internal.i := 0 TO MAX_ITEM_X_IDX DO
		// Find Next Lowest Index
		Internal.tempIndex							:= Internal.i;
		IF ItemX.List[Internal.tempIndex].UID = 0 THEN
			Internal.tempUID						:= 4294967295; // Set to UDINT max
		ELSE
			Internal.tempUID						:= ItemX.List[Internal.tempIndex].UID;
		END_IF;
		FOR Internal.j := Internal.i TO MAX_ITEM_X_IDX DO
			IF ItemX.List[Internal.j].UID < Internal.tempUID AND ItemX.List[Internal.j].UID > 0 THEN
				Internal.tempIndex					:= Internal.j;
				Internal.tempUID					:= ItemX.List[Internal.tempIndex].UID;
			END_IF;
		END_FOR;
		// Swap ItemXs
		Internal.tempItemX							:= ItemX.List[Internal.i];
		ItemX.List[Internal.i]						:= ItemX.List[Internal.tempIndex];
		ItemX.List[Internal.tempIndex]				:= Internal.tempItemX;
		IF ItemX.List[Internal.i].UID = 0 THEN
			ItemX.ReturnedIndex 						:= Internal.i;
			EXIT;
		END_IF;
	END_FOR;

	// This is here for keeping the ItemX structure up to date and should be at the bottom of every function call in the library
	ItemX.ValidIndex									:= FALSE;
	IF ItemX.ReturnedIndex >= 0 AND ItemX.ReturnedIndex <= MAX_ITEM_X_IDX THEN
		ItemX.ValidIndex								:= TRUE;
	END_IF;

END_FUNCTION
```

#### TC_ItemX_Sanitize.st
```iecst
(* Deletes all ItemXs that have UID of 0 *)
FUNCTION TC_ItemX_Sanitize
	TC_ItemX_Sanitize								:= TRUE;
	FOR Internal.i := 0 TO MAX_ITEM_X_IDX DO
		IF ItemX.List[Internal.i].UID = 0 THEN
			brsmemset(ADR(ItemX.List[Internal.i]),0,SIZEOF(ItemX.List[Internal.i]));
		END_IF;
	END_FOR;

	TC_ItemX_FirstOpenIndex(ItemX);
	// This is here for keeping the ItemX structure up to date and should be at the bottom of every function call in the library
	ItemX.ValidIndex									:= FALSE;
	IF ItemX.ReturnedIndex >= 0 AND ItemX.ReturnedIndex <= MAX_ITEM_X_IDX THEN
		ItemX.ValidIndex								:= TRUE;
	END_IF;

END_FUNCTION
```

#### TC_ItemX_IncrementUID.st
```iecst
(* IncrementsUID, Ensures that the UID will be the Highest in the list if it isnt *)
FUNCTION TC_ItemX_IncrementUID
	TC_ItemX_IncrementUID							:= TRUE;
	ItemX.CurrentUID								:= ItemX.CurrentUID + 1;

	Internal.tempUID								:= 0;
	FOR Internal.i := 0 TO MAX_ITEM_X_IDX DO
		IF ItemX.List[Internal.i].UID > Internal.tempUID THEN
			Internal.tempUID						:= ItemX.List[Internal.i].UID;
		END_IF;
	END_FOR;
	IF Internal.tempUID >= ItemX.CurrentUID THEN
		ItemX.CurrentUID							:= Internal.tempUID + 1;
	END_IF;

	// This is here for keeping the ItemX structure up to date and should be at the bottom of every function call in the library
	ItemX.ValidIndex								:= FALSE;
	IF ItemX.ReturnedIndex >= 0 AND ItemX.ReturnedIndex <= MAX_ITEM_X_IDX THEN
		ItemX.ValidIndex							:= TRUE;
	END_IF;

END_FUNCTION
```

#### TC_ItemX_AddElem.st
```iecst
(* Adds Elem to List, returns true if successful and changes index to where it was added *)
FUNCTION TC_ItemX_AddElem

	TC_ItemX_AddElem								:= FALSE;
	ItemX.ReturnedIndex								:= -1;
	FOR Internal.i := 0 TO MAX_ITEM_X_IDX DO
		IF ItemX.List[Internal.i].UID = 0 THEN
			TC_ItemX_AddElem						:= TRUE;
			ItemX.ReturnedIndex						:= Internal.i;
			TC_ItemX_IncrementUID(ItemX);
			ItemX.Elem.UID							:= ItemX.CurrentUID;
			ItemX.List[Internal.i]					:= ItemX.Elem;
			EXIT;
		END_IF;
	END_FOR;

	// This is here for keeping the ItemX structure up to date and should be at the bottom of every function call in the library
	ItemX.ValidIndex								:= FALSE;
	IF ItemX.ReturnedIndex >= 0 AND ItemX.ReturnedIndex <= MAX_ITEM_X_IDX THEN
		ItemX.ValidIndex							:= TRUE;
	END_IF;

END_FUNCTION
```

#### TC_ItemX_ModElemByUID.st
```iecst
(* Modifies Elem in List without changing UID, returns true if successful *)
FUNCTION TC_ItemX_ModElemByUID

	TC_ItemX_ModElemByUID							:= FALSE;
	ItemX.ReturnedIndex								:= -1;

	FOR Internal.i := 0 TO MAX_ITEM_X_IDX DO
		IF ItemX.List[Internal.i].UID = UID THEN
			ItemX.Elem.UID							:= UID;
			ItemX.List[Internal.i]					:= ItemX.Elem;
			ItemX.List[Internal.i].UID 				:= UID;
			ItemX.ReturnedIndex						:= Internal.i;
			TC_ItemX_ModElemByUID					:= TRUE;
			EXIT;
		END_IF;
	END_FOR;

	// This is here for keeping the ItemX structure up to date and should be at the bottom of every function call in the library
	ItemX.ValidIndex								:= FALSE;
	IF ItemX.ReturnedIndex >= 0 AND ItemX.ReturnedIndex <= MAX_ITEM_X_IDX THEN
		ItemX.ValidIndex							:= TRUE;
	END_IF;

END_FUNCTION
```

#### TC_ItemX_ModElemByIndex.st
```iecst
(* Modifies Elem in List without changing UID, returns true if successful *)
FUNCTION TC_ItemX_ModElemByIndex

	TC_ItemX_ModElemByIndex							:= FALSE;
	ItemX.ReturnedIndex								:= -1;

	IF Index >= 0 AND Index <= MAX_ITEM_X_IDX THEN
		IF ItemX.List[Index].UID = 0 THEN
			TC_ItemX_AddElem(ItemX);
		ELSE
			Internal.tempUID						:= ItemX.List[Index].UID;
			ItemX.List[Index]						:= ItemX.Elem;
			ItemX.List[Internal.i].UID 				:= Internal.tempUID;
		END_IF;
		ItemX.ReturnedIndex							:= Index;
		TC_ItemX_ModElemByIndex						:= TRUE;
	END_IF;

	// This is here for keeping the ItemX structure up to date and should be at the bottom of every function call in the library
	ItemX.ValidIndex								:= FALSE;
	IF ItemX.ReturnedIndex >= 0 AND ItemX.ReturnedIndex <= MAX_ITEM_X_IDX THEN
		ItemX.ValidIndex							:= TRUE;
	END_IF;

END_FUNCTION
```

#### TC_ItemX_GetElemByUID.st
```iecst
(* Gets Elem in List, returns true if successful *)
FUNCTION TC_ItemX_GetElemByUID

	TC_ItemX_GetElemByUID							:= FALSE;
	ItemX.ReturnedIndex								:= -1;

	FOR Internal.i := 0 TO MAX_ITEM_X_IDX DO
		IF ItemX.List[Internal.i].UID = UID THEN
			ItemX.Elem								:= ItemX.List[Internal.i];
			ItemX.ReturnedIndex						:= Internal.i;
			TC_ItemX_GetElemByUID					:= TRUE;
			EXIT;
		END_IF;
	END_FOR;

	// This is here for keeping the ItemX structure up to date and should be at the bottom of every function call in the library
	ItemX.ValidIndex								:= FALSE;
	IF ItemX.ReturnedIndex >= 0 AND ItemX.ReturnedIndex <= MAX_ITEM_X_IDX THEN
		ItemX.ValidIndex							:= TRUE;
	END_IF;

END_FUNCTION
```

#### TC_ItemX_GetElemByIndex.st
```iecst
(* Gets Elem in List, returns true if successful *)
FUNCTION TC_ItemX_GetElemByIndex
	Internal.i 										:= 0; // This is to avoid a compiler warning that internal is not used.
	TC_ItemX_GetElemByIndex							:= FALSE;
	ItemX.ReturnedIndex								:= -1;

	IF Index >= 0 AND Index <= MAX_ITEM_X_IDX THEN
		IF ItemX.List[Index].UID <> 0 THEN
			ItemX.Elem								:= ItemX.List[Index];
			ItemX.ReturnedIndex						:= Index;
			TC_ItemX_GetElemByIndex					:= TRUE;
		END_IF;
	END_IF;

	// This is here for keeping the ItemX structure up to date and should be at the bottom of every function call in the library
	ItemX.ValidIndex								:= FALSE;
	IF ItemX.ReturnedIndex >= 0 AND ItemX.ReturnedIndex <= MAX_ITEM_X_IDX THEN
		ItemX.ValidIndex							:= TRUE;
	END_IF;

END_FUNCTION
```

### Library Logical/Libraries/TC_Array (IEC)
Depends on: AsBrStr

#### Constants.var - Exported constants
```iecst
VAR CONSTANT
	TC_ARRAY_MAXELEMENTSIZE : UINT := 2000;
END_VAR
```

#### TC_Array.fun - Exported functions and function blocks
```iecst
{REDUND_ERROR} FUNCTION TC_Array_PeekTop : INT (*Peeks at the top index of an array without removing it*) (*$GROUP=User,$CAT=User,$GROUPICON=User.png,$CATICON=User.png*)
	VAR_INPUT
		pBuffer : UDINT;
		sizeBuffer : UDINT;
		pElement : UDINT;
		SizeElement : UDINT;
	END_VAR
	VAR
		emptyData : ARRAY[0..TC_ARRAY_MAXELEMENTSIZE] OF USINT;
		i : UDINT;
	END_VAR
END_FUNCTION

{REDUND_ERROR} FUNCTION TC_Array_AddTop : INT (*Adds the first index of an array*) (*$GROUP=User,$CAT=User,$GROUPICON=User.png,$CATICON=User.png*)
	VAR_INPUT
		pBuffer : UDINT;
		SizeBuffer : UDINT;
		pElement : UDINT;
		SizeElement : UDINT;
	END_VAR
END_FUNCTION

{REDUND_ERROR} FUNCTION TC_Array_AddBottom : BOOL (*Removes the last index of an array*) (*$GROUP=User,$CAT=User,$GROUPICON=User.png,$CATICON=User.png*)
	VAR_INPUT
		pBuffer : UDINT;
		SizeBuffer : UDINT;
		pElement : UDINT;
		SizeElement : UDINT;
	END_VAR
END_FUNCTION

{REDUND_ERROR} FUNCTION TC_Array_PeekBtm : INT (*Copies the last index in an array to the output without removing it*) (*$GROUP=User,$CAT=User,$GROUPICON=User.png,$CATICON=User.png*)
	VAR_INPUT
		pBuffer : UDINT;
		sizeBuffer : UDINT;
		pElement : UDINT;
		SizeElement : UDINT;
	END_VAR
	VAR
		emptyData : ARRAY[0..TC_ARRAY_MAXELEMENTSIZE] OF USINT;
		i : DINT;
	END_VAR
END_FUNCTION

{REDUND_ERROR} FUNCTION TC_Array_Pop : INT (*Pops the top index out of the array into out variable*) (*$GROUP=User,$CAT=User,$GROUPICON=User.png,$CATICON=User.png*)
	VAR_INPUT
		pBuffer : UDINT;
		sizeBuffer : UDINT;
		pElement : UDINT;
		SizeElement : UDINT;
	END_VAR
	VAR
		emptyData : ARRAY[0..TC_ARRAY_MAXELEMENTSIZE] OF USINT;
		i : UDINT;
		nextSpot : UDINT;
	END_VAR
END_FUNCTION

{REDUND_ERROR} FUNCTION TC_Array_Dequeue : INT (*Dequeues the last index in an array to the output*) (*$GROUP=User,$CAT=User,$GROUPICON=User.png,$CATICON=User.png*)
	VAR_INPUT
		pBuffer : UDINT;
		sizeBuffer : UDINT;
		pElement : UDINT;
		SizeElement : UDINT;
	END_VAR
	VAR
		emptyData : ARRAY[0..TC_ARRAY_MAXELEMENTSIZE] OF USINT;
		i : DINT;
	END_VAR
END_FUNCTION

{REDUND_ERROR} FUNCTION TC_Array_Pack : INT (*TODO: Add your comment here*) (*$GROUP=User,$CAT=User,$GROUPICON=User.png,$CATICON=User.png*)
	VAR_INPUT
		pBuffer : UDINT;
		sizeBuffer : UDINT;
		SizeElement : UDINT;
	END_VAR
	VAR
		emptyData : ARRAY[0..TC_ARRAY_MAXELEMENTSIZE] OF USINT;
		i : UDINT;
		dataFound : UDINT;
	END_VAR
END_FUNCTION
```

#### TC_Array_AddTop.st
```iecst
(* Adds the first index of an array *)
FUNCTION TC_Array_AddTop

	TC_Array_AddTop := 0;

	//Input Error Checking
	IF 	pBuffer = 0 THEN
		TC_Array_AddTop.15 := 1;
		TC_Array_AddTop.0  := 1;
	END_IF

	IF pElement = 0 THEN
		TC_Array_AddTop.15 := 1;
		TC_Array_AddTop.1  := 1;
	END_IF

	IF SizeBuffer = 0 THEN
		TC_Array_AddTop.15 := 1;
		TC_Array_AddTop.2  := 1;
	END_IF

	IF SizeElement = 0 THEN
		TC_Array_AddTop.15 := 1;
		TC_Array_AddTop.3  := 1;
	END_IF

	IF SizeBuffer < SizeElement * 2 THEN
		TC_Array_AddTop.15 := 1;
		TC_Array_AddTop.4  := 1;
	END_IF

	IF SizeBuffer MOD SizeElement <> 0 THEN
		TC_Array_AddTop.15 := 1;
		TC_Array_AddTop.5  := 1;
	END_IF

	IF TC_Array_AddTop = 0 THEN
		//Everything passed we can go to work
		brsmemmove(pBuffer + SizeElement, pBuffer, SizeBuffer - SizeElement);
		brsmemcpy(pBuffer, pElement, SizeElement);
	END_IF

END_FUNCTION
```

#### TC_Array_AddBottom.st
```iecst
(* Removes the last index of an array *)
FUNCTION TC_Array_AddBottom
	pBuffer;
	SizeBuffer;
	pElement;
	SizeElement;
	TC_Array_AddBottom := TRUE;
END_FUNCTION
```

#### TC_Array_PeekTop.st
```iecst
(* Peeks at the top index of an array without removing it *)
FUNCTION TC_Array_PeekTop

	TC_Array_PeekTop := 0;
	brsmemset(ADR(emptyData), 0, SIZEOF(emptyData));

	//Validate input parameters
	IF pBuffer = 0 THEN
		TC_Array_PeekTop.0  := TRUE;
		TC_Array_PeekTop.15 := TRUE;
	END_IF

	IF sizeBuffer = 0 THEN
		TC_Array_PeekTop.1  := TRUE;
		TC_Array_PeekTop.15 := TRUE;
	END_IF

	IF pElement = 0 THEN
		TC_Array_PeekTop.2  := TRUE;
		TC_Array_PeekTop.15 := TRUE;
	END_IF

	IF SizeElement = 0 THEN
		TC_Array_PeekTop.3  := TRUE;
		TC_Array_PeekTop.15 := TRUE;
	END_IF

	IF sizeBuffer MOD SizeElement <> 0 THEN
		TC_Array_PeekTop.4  := TRUE;
		TC_Array_PeekTop.15 := TRUE;
	END_IF

	IF SizeElement > TC_ARRAY_MAXELEMENTSIZE THEN
		TC_Array_PeekTop.5  := TRUE;
		TC_Array_PeekTop.15 := TRUE;
	END_IF

	//Everything passed we can go a head and peek
	IF TC_Array_PeekTop = 0 THEN
		FOR i:=0 TO (sizeBuffer / SizeElement)-1 DO
			IF brsmemcmp(pBuffer + SizeElement*i, ADR(emptyData), SizeElement) <> 0 THEN
				//We found the first index
				brsmemcpy(pElement, pBuffer + SizeElement*i, SizeElement);
				TC_Array_PeekTop := 1;
				EXIT;
			END_IF
		END_FOR
	END_IF

END_FUNCTION
```

#### TC_Array_PeekBtm.st
```iecst
(*Peeks at the bottom of the array without moving it.. cheeky monkey
	Returns (-) number for error, 0 for nothing in array and 1 when it finds something*)
FUNCTION TC_Array_PeekBtm

	TC_Array_PeekBtm := 0;
	brsmemset(ADR(emptyData), 0, SIZEOF(emptyData));

	//Validate input parameters
	IF pBuffer = 0 THEN
		TC_Array_PeekBtm.0  := TRUE;
		TC_Array_PeekBtm.15 := TRUE;
	END_IF

	IF sizeBuffer = 0 THEN
		TC_Array_PeekBtm.1  := TRUE;
		TC_Array_PeekBtm.15 := TRUE;
	END_IF

	IF pElement = 0 THEN
		TC_Array_PeekBtm.2  := TRUE;
		TC_Array_PeekBtm.15 := TRUE;
	END_IF

	IF SizeElement = 0 THEN
		TC_Array_PeekBtm.3  := TRUE;
		TC_Array_PeekBtm.15 := TRUE;
	END_IF

	IF sizeBuffer MOD SizeElement <> 0 THEN
		TC_Array_PeekBtm.4  := TRUE;
		TC_Array_PeekBtm.15 := TRUE;
	END_IF

	IF SizeElement > TC_ARRAY_MAXELEMENTSIZE THEN
		TC_Array_PeekBtm.5  := TRUE;
		TC_Array_PeekBtm.15 := TRUE;
	END_IF

	//Everything passed we can go a head and peek
	IF TC_Array_PeekBtm = 0 THEN
		FOR i:= (sizeBuffer / SizeElement)-1 TO 0 BY -1 DO
			IF brsmemcmp(pBuffer + SizeElement*DINT_TO_UDINT(i), ADR(emptyData), SizeElement) <> 0 THEN
				//We found the first index
				brsmemcpy(pElement, pBuffer + SizeElement*DINT_TO_UDINT(i), SizeElement);
				TC_Array_PeekBtm := 1;
				EXIT;
			END_IF
		END_FOR
	END_IF

END_FUNCTION
```

#### TC_Array_Pop.st
```iecst
(* Pops the top index out of the array into out variable *)
FUNCTION TC_Array_Pop

	TC_Array_Pop := 0;
	brsmemset(ADR(emptyData), 0, SIZEOF(emptyData));

	//Validate input parameters
	IF pBuffer = 0 THEN
		TC_Array_Pop.0  := TRUE;
		TC_Array_Pop.15 := TRUE;
	END_IF

	IF sizeBuffer = 0 THEN
		TC_Array_Pop.1  := TRUE;
		TC_Array_Pop.15 := TRUE;
	END_IF

	IF pElement = 0 THEN
		TC_Array_Pop.2  := TRUE;
		TC_Array_Pop.15 := TRUE;
	END_IF

	IF SizeElement = 0 THEN
		TC_Array_Pop.3  := TRUE;
		TC_Array_Pop.15 := TRUE;
	END_IF

	IF sizeBuffer MOD SizeElement <> 0 THEN
		TC_Array_Pop.4  := TRUE;
		TC_Array_Pop.15 := TRUE;
	END_IF

	IF SizeElement > TC_ARRAY_MAXELEMENTSIZE THEN
		TC_Array_Pop.5  := TRUE;
		TC_Array_Pop.15 := TRUE;
	END_IF

	//Everything passed we can go a head and look for an index to pop
	IF TC_Array_Pop = 0 THEN
		FOR i:=0 TO (sizeBuffer / SizeElement) - 1 DO
			IF brsmemcmp(pBuffer + SizeElement*i, ADR(emptyData), SizeElement) <> 0 THEN
				//We found the first index
				brsmemcpy(pElement, pBuffer + SizeElement*i, SizeElement);
				nextSpot := brsmemmove(pBuffer, pBuffer + SizeElement*(i+1), sizeBuffer - SizeElement * (i+1));
				brsmemset(nextSpot, 0, SizeElement*(i+1));
				TC_Array_Pop := 1;
				EXIT;
			END_IF
		END_FOR
	END_IF

END_FUNCTION
```

#### TC_Array_Dequeue.st
```iecst
(* Dequeues the last index in an array to the output *)
FUNCTION TC_Array_Dequeue

	TC_Array_Dequeue := 0;
	brsmemset(ADR(emptyData), 0, SIZEOF(emptyData));

	//Validate input parameters
	IF pBuffer = 0 THEN
		TC_Array_Dequeue.0  := TRUE;
		TC_Array_Dequeue.15 := TRUE;
	END_IF

	IF sizeBuffer = 0 THEN
		TC_Array_Dequeue.1  := TRUE;
		TC_Array_Dequeue.15 := TRUE;
	END_IF

	IF pElement = 0 THEN
		TC_Array_Dequeue.2  := TRUE;
		TC_Array_Dequeue.15 := TRUE;
	END_IF

	IF SizeElement = 0 THEN
		TC_Array_Dequeue.3  := TRUE;
		TC_Array_Dequeue.15 := TRUE;
	END_IF

	IF sizeBuffer MOD SizeElement <> 0 THEN
		TC_Array_Dequeue.4  := TRUE;
		TC_Array_Dequeue.15 := TRUE;
	END_IF

	IF SizeElement > TC_ARRAY_MAXELEMENTSIZE THEN
		TC_Array_Dequeue.5  := TRUE;
		TC_Array_Dequeue.15 := TRUE;
	END_IF

	//Everything passed we can go a head and peek
	IF TC_Array_Dequeue = 0 THEN
		FOR i:= (sizeBuffer / SizeElement) - 1 TO 0 BY -1 DO
			IF brsmemcmp(pBuffer + SizeElement*DINT_TO_UDINT(i), ADR(emptyData), SizeElement) <> 0 THEN
				//We found the first index
				brsmemcpy(pElement, pBuffer + SizeElement*DINT_TO_UDINT(i), SizeElement);
				brsmemset(pBuffer + SizeElement*DINT_TO_UDINT(i), 0, SizeElement);
				TC_Array_Dequeue := 1;
				EXIT;
			END_IF
		END_FOR
	END_IF

END_FUNCTION
```

#### TC_Array_Pack.st
```iecst
(* TODO: Actually make this work *)
FUNCTION TC_Array_Pack

	TC_Array_Pack := 0;
	brsmemset(ADR(emptyData), 0, SIZEOF(emptyData));

	//Validate input parameters
	IF pBuffer = 0 THEN
		TC_Array_Pack.0  := TRUE;
		TC_Array_Pack.15 := TRUE;
	END_IF

	IF sizeBuffer = 0 THEN
		TC_Array_Pack.1  := TRUE;
		TC_Array_Pack.15 := TRUE;
	END_IF

	IF TC_Array_Pack = 0 THEN
		FOR i:= (sizeBuffer / SizeElement) TO 1 BY -1 DO
			IF brsmemcmp(pBuffer + SizeElement*i, ADR(emptyData), SizeElement) = 0 THEN
				IF dataFound <> 0 THEN
					brsmemmove(pBuffer + SizeElement*i, pBuffer + SizeElement*(i+1), dataFound*SizeElement);
				END_IF
			ELSE
				dataFound := dataFound + 1;
			END_IF
		END_FOR
	END_IF

END_FUNCTION
```

### Library Logical/Libraries/TC_SysErr (IEC, version 1.0.0)
Depends on: ArTextSys, AsBrStr, ArEventLog

#### Types.typ - Exported data types
```iecst
TYPE
	Internal_TC_SysErr_Log : 	STRUCT
		State : INT;
		TC_SysErr_Lookup_0 : TC_SysErr_Lookup;
		ArEventLogGetIdent_0 : ArEventLogGetIdent;
		ArEventLogWrite_0 : ArEventLogWrite;
		AddData : STRING[255];
	END_STRUCT;
	Internal_TC_SysErr_Lookup : 	STRUCT
		ArTextSysGetText_0 : ArTextSysGetText;
		TextID : STRING[255];
		ErrorNumString : STRING[80];
		State : INT;
	END_STRUCT;
END_TYPE
```

#### TC_SysErr.fun - Exported functions and function blocks
```iecst
{REDUND_ERROR} FUNCTION_BLOCK TC_SysErr_Lookup (*Returns System Error If It Exists In Table*) (*$GROUP=User,$CAT=User,$GROUPICON=User.png,$CATICON=User.png*)
	VAR_INPUT
		Execute : BOOL;
		ErrorNum : DINT;
	END_VAR
	VAR_OUTPUT
		ErrorNumText : STRING[255];
		Error : BOOL;
		Done : BOOL;
	END_VAR
	VAR
		Internal : Internal_TC_SysErr_Lookup;
	END_VAR
END_FUNCTION_BLOCK

{REDUND_ERROR} FUNCTION_BLOCK TC_SysErr_Log (*Returns System Error If It Exists In Table*) (*$GROUP=User,$CAT=User,$GROUPICON=User.png,$CATICON=User.png*)
	VAR_INPUT
		Execute : BOOL;
		ErrorNum : DINT;
	END_VAR
	VAR_OUTPUT
		ErrorNumText : STRING[255];
		Error : BOOL;
		Done : BOOL;
	END_VAR
	VAR
		Internal : Internal_TC_SysErr_Log;
	END_VAR
END_FUNCTION_BLOCK
```

#### TC_SysErr_Lookup.st
```iecst
(* Returns System Error If It Exists In Table *)
FUNCTION_BLOCK TC_SysErr_Lookup

	IF NOT Execute THEN
		Internal.State := 0;
	END_IF;
	CASE Internal.State OF
		0:
			brsmemset(ADR(ErrorNumText),0,SIZEOF(ErrorNumText));
			Internal.ArTextSysGetText_0.Execute := FALSE;
			Error := FALSE;
			Done := FALSE;
			IF Execute THEN
				Internal.State := 10;
			END_IF;
		10:
			brsmemset(ADR(ErrorNumText),0,SIZEOF(ErrorNumText));
			brsmemset(ADR(Internal.TextID),0,SIZEOF(Internal.TextID));
			brsmemset(ADR(Internal.ErrorNumString),0,SIZEOF(Internal.ErrorNumString));
			brsitoa(ErrorNum,ADR(Internal.ErrorNumString));
			brsstrcat(ADR(Internal.TextID),ADR('TC_SysErr.'));
			brsstrcat(ADR(Internal.TextID),ADR(Internal.ErrorNumString));
			Internal.ArTextSysGetText_0.Execute := TRUE;
			Internal.State := 20;
		20:
			IF Internal.ArTextSysGetText_0.Done THEN
				Done := TRUE;
				Internal.State := 30;
			ELSIF Internal.ArTextSysGetText_0.Error THEN
				Error := TRUE;
				Internal.State := 30;
			END_IF;
		30:
			IF Error THEN
				ErrorNumText := 'Not Found';
			END_IF;
	END_CASE;
	Internal.ArTextSysGetText_0(Namespace := ADR('TC_SysErr'), TextID := ADR(Internal.TextID), LanguageCode := 'en', TextBufferSize := SIZEOF(ErrorNumText)-1, TextBuffer := ADR(ErrorNumText), SearchMode := arTEXTSYS_SEARCH_LANGUAGE_ONLY);

END_FUNCTION_BLOCK
```

#### TC_SysErr_Log.st
```iecst
(* Returns System Error If It Exists In Table and Logs it to the user logger*)
FUNCTION_BLOCK TC_SysErr_Log
	IF NOT Execute THEN
		Internal.State := 0;
	END_IF;
	CASE Internal.State OF
		0:
			brsmemset(ADR(ErrorNumText),0,SIZEOF(ErrorNumText));
			Internal.TC_SysErr_Lookup_0.Execute := FALSE;
			Error := FALSE;
			Done := FALSE;
			IF Execute THEN
				Internal.State := 10;
			END_IF;
		10:
			brsmemset(ADR(ErrorNumText),0,SIZEOF(ErrorNumText));
			Internal.TC_SysErr_Lookup_0.ErrorNum := ErrorNum;
			Internal.TC_SysErr_Lookup_0.Execute := TRUE;
			Internal.State := 20;
		20:
			IF Internal.TC_SysErr_Lookup_0.Done THEN
				ErrorNumText := Internal.TC_SysErr_Lookup_0.ErrorNumText;
				Internal.State := 100;
			ELSIF Internal.TC_SysErr_Lookup_0.Error THEN
				ErrorNumText := Internal.TC_SysErr_Lookup_0.ErrorNumText;
				Internal.State := 99;
			END_IF;
		99:
			Error := TRUE;
		100:
			brsmemset(ADR(Internal.AddData),0,SIZEOF(Internal.AddData));
			brsstrcat(ADR(Internal.AddData),ADR(ErrorNumText));
			Internal.ArEventLogGetIdent_0.Name := '$$arlogusr';
			Internal.ArEventLogGetIdent_0.Execute := TRUE;
			Internal.State := 110;
		110:
			IF Internal.ArEventLogGetIdent_0.Done THEN
				Internal.ArEventLogGetIdent_0.Execute := FALSE;
				Internal.ArEventLogWrite_0.Ident := Internal.ArEventLogGetIdent_0.Ident;
				Internal.ArEventLogWrite_0.EventID := -536870912;
				Internal.ArEventLogWrite_0.ObjectID := 'TC_SysErr';
				Internal.ArEventLogWrite_0.AddDataFormat := 1;
				Internal.ArEventLogWrite_0.AddData := ADR(Internal.AddData);
				Internal.ArEventLogWrite_0.AddDataSize := brsstrlen(ADR(Internal.AddData))+1;
				Internal.ArEventLogWrite_0.Execute := TRUE;
				Internal.State := 120;
			ELSIF Internal.ArEventLogGetIdent_0.Error THEN
				Internal.State := 999;
			END_IF;
		120:
			IF Internal.ArEventLogWrite_0.Done THEN
				Internal.ArEventLogWrite_0.Execute := FALSE;
				Internal.State := 130;
			ELSIF NOT Internal.ArEventLogWrite_0.Error THEN
				Internal.State := 999;
			END_IF;
		130:
			Done := TRUE;
		999:
			Error := TRUE;
			ErrorNumText := 'Log Error';
	END_CASE;
	Internal.TC_SysErr_Lookup_0();
	Internal.ArEventLogGetIdent_0();
	Internal.ArEventLogWrite_0();
END_FUNCTION_BLOCK
```

### Library Logical/Libraries/TC_Eval (IEC)

#### Types.typ - Exported data types
```iecst
TYPE
	TC_Eval_Internal_typ : 	STRUCT
		CTON_DB_Off : CTON;
		CTON_DB_On : CTON;
		StatusResult : BOOL;
		i : DINT;
	END_STRUCT;
	TC_Eval_Sim_typ : 	STRUCT
		Active : BOOL;
		Logical : BOOL;
	END_STRUCT;
	TC_Eval_Signal_typ : 	STRUCT
		Logical : BOOL;
		Result : BOOL;
		EdgePosResult : BOOL;
		EdgeNegResult : BOOL;
	END_STRUCT;
	TC_Eval_Par_typ : 	STRUCT
		FilterOnTime : LREAL;
		FilterOffTime : LREAL;
	END_STRUCT;
	TC_Eval_Forcing_typ : 	STRUCT
		Off : BOOL;
		On : BOOL;
	END_STRUCT;
	TC_EVAL_OPERATOR_ENUM :
		(
		TC_EVAL_OP_AND,
		TC_EVAL_OP_OR
		);
END_TYPE
```

#### Constants.var - Exported constants
```iecst
VAR CONSTANT
	MAX_EVAL_LOGICAL_IDX : DINT := 4;
END_VAR
```

#### TC_Eval.fun - Exported functions and function blocks
```iecst
{REDUND_ERROR} FUNCTION_BLOCK TC_Eval (*Evalditional Handler*) (*$GROUP=User,$CAT=User,$GROUPICON=User.png,$CATICON=User.png*)
	VAR_INPUT
		ES_ID : STRING[32];
		Logical : ARRAY[0..MAX_EVAL_LOGICAL_IDX] OF BOOL;
		Operator : TC_EVAL_OPERATOR_ENUM;
		Call : DINT;
		ES_Call : STRING[32];
		Par : TC_Eval_Par_typ;
		Forcing : TC_Eval_Forcing_typ;
		Sim : TC_Eval_Sim_typ;
		EdgeReset : BOOL;
	END_VAR
	VAR_OUTPUT
		Signal : TC_Eval_Signal_typ;
	END_VAR
	VAR
		Internal : TC_Eval_Internal_typ;
	END_VAR
END_FUNCTION_BLOCK
```

#### TC_Eval.st
```iecst
FUNCTION_BLOCK TC_Eval
//Usage for warning supression
	ES_ID;
	ES_Call;
	Call;
//Interaction
	IF Forcing.Off THEN
		Signal.Logical					:= FALSE;
	ELSIF Forcing.On THEN
		Signal.Logical					:= TRUE;
	ELSIF Sim.Active THEN
		Signal.Logical					:= Sim.Logical;
	ELSIF Operator = TC_EVAL_OP_AND THEN
		Signal.Logical					:= TRUE;
		FOR Internal.i := 0 TO MAX_EVAL_LOGICAL_IDX DO
			IF NOT Logical[Internal.i] THEN
				Signal.Logical			:= FALSE;
				EXIT;
			END_IF;
		END_FOR;
	ELSIF Operator = TC_EVAL_OP_OR THEN
		Signal.Logical					:= FALSE;
		FOR Internal.i := 0 TO MAX_EVAL_LOGICAL_IDX DO
			IF Logical[Internal.i] THEN
				Signal.Logical			:= TRUE;
				EXIT;
			END_IF;
		END_FOR;
	ELSE
		Signal.Logical					:= FALSE;
	END_IF;
//Debouncing
	IF Signal.Logical THEN
		Internal.CTON_DB_Off(IN := FALSE);
		Internal.CTON_DB_On(IN := TRUE, PT := LREAL_TO_TIME(Par.FilterOnTime*1000.0));
		IF Internal.CTON_DB_On.Q OR Par.FilterOnTime <= 0.0 THEN
			Signal.Result				:= TRUE;
		END_IF;
	ELSE
		Internal.CTON_DB_On(IN := FALSE);
		Internal.CTON_DB_Off(IN := TRUE, PT := LREAL_TO_TIME(Par.FilterOffTime*1000.0));
		IF Internal.CTON_DB_Off.Q OR Par.FilterOffTime <= 0.0 THEN
			Signal.Result				:= FALSE;
		END_IF;
	END_IF;
//Edges
	IF EdgeReset THEN
		Signal.EdgePosResult			:= FALSE;
		Signal.EdgeNegResult			:= FALSE;
		Internal.StatusResult			:= FALSE;
	ELSE
		Signal.EdgeNegResult			:= FALSE;
		IF Internal.StatusResult AND NOT Signal.Result THEN
			Signal.EdgeNegResult		:= TRUE;
		END_IF;
		Signal.EdgePosResult			:= FALSE;
		IF NOT Internal.StatusResult AND Signal.Result THEN
			Signal.EdgePosResult		:= TRUE;
		END_IF;
		Internal.StatusResult 			:= Signal.Result;
	END_IF;
END_FUNCTION_BLOCK
```

### Library Logical/Libraries/TC_Mon (IEC)

#### Types.typ - Exported data types
```iecst
TYPE
	TC_Mon_Internal_typ : 	STRUCT
		CTON_DB_Off : CTON;
		CTON_DB_On : CTON;
		StatusResult : BOOL;
		i : DINT;
	END_STRUCT;
	TC_Mon_ProcessMask_typ : 	STRUCT
		Sev : DINT;
		ES_ID : STRING[32];
	END_STRUCT;
	TC_Mon_Sim_typ : 	STRUCT
		Active : BOOL;
		Logical : BOOL;
	END_STRUCT;
	TC_Mon_Signal_typ : 	STRUCT
		Logical : BOOL;
		Result : BOOL;
		EdgePosResult : BOOL;
		EdgeNegResult : BOOL;
	END_STRUCT;
	TC_Mon_Par_typ : 	STRUCT
		FilterOnTime : LREAL;
		FilterOffTime : LREAL;
	END_STRUCT;
	TC_Mon_Forcing_typ : 	STRUCT
		Off : BOOL;
		On : BOOL;
	END_STRUCT;
	TC_MON_OPERATOR_ENUM :
		(
		TC_MON_OP_AND,
		TC_MON_OP_OR
		);
END_TYPE
```

#### Constants.var - Exported constants
```iecst
VAR CONSTANT
	MAX_TC_MON_PROCESS_IDX : DINT := 2;
	MAX_MON_LOGICAL_IDX : DINT := 4;
END_VAR
```

#### TC_Mon.fun - Exported functions and function blocks
```iecst
{REDUND_ERROR} FUNCTION_BLOCK TC_Mon (*Conditional Handler*) (*$GROUP=User,$CAT=User,$GROUPICON=User.png,$CATICON=User.png*)
	VAR_INPUT
		ES_ID : STRING[32];
		Operator : TC_MON_OPERATOR_ENUM;
		Logical : ARRAY[0..MAX_MON_LOGICAL_IDX] OF BOOL;
		Sev : DINT;
		Mask : ARRAY[0..MAX_TC_MON_PROCESS_IDX] OF TC_Mon_ProcessMask_typ;
		Par : TC_Mon_Par_typ;
		Forcing : TC_Mon_Forcing_typ;
		Sim : TC_Mon_Sim_typ;
		EdgeReset : BOOL;
	END_VAR
	VAR_OUTPUT
		Signal : TC_Mon_Signal_typ;
	END_VAR
	VAR
		Internal : TC_Mon_Internal_typ;
	END_VAR
END_FUNCTION_BLOCK
```

#### TC_Mon.st
```iecst
FUNCTION_BLOCK TC_Mon
//Usage for warning supression
	ES_ID;
	Sev;
	Mask;
//Interaction
	IF Forcing.Off THEN
		Signal.Logical					:= FALSE;
	ELSIF Forcing.On THEN
		Signal.Logical					:= TRUE;
	ELSIF Sim.Active THEN
		Signal.Logical					:= Sim.Logical;
	ELSIF Operator = TC_MON_OP_AND THEN
		Signal.Logical					:= TRUE;
		FOR Internal.i := 0 TO MAX_MON_LOGICAL_IDX DO
			IF NOT Logical[Internal.i] THEN
				Signal.Logical			:= FALSE;
				EXIT;
			END_IF;
		END_FOR;
	ELSIF Operator = TC_MON_OP_OR THEN
		Signal.Logical					:= FALSE;
		FOR Internal.i := 0 TO MAX_MON_LOGICAL_IDX DO
			IF Logical[Internal.i] THEN
				Signal.Logical			:= TRUE;
				EXIT;
			END_IF;
		END_FOR;
	ELSE
		Signal.Logical					:= FALSE;
	END_IF;
//Debouncing
	IF Signal.Logical THEN
		Internal.CTON_DB_Off(IN := FALSE);
		Internal.CTON_DB_On(IN := TRUE, PT := LREAL_TO_TIME(Par.FilterOnTime*1000.0));
		IF Internal.CTON_DB_On.Q OR Par.FilterOnTime <= 0.0 THEN
			Signal.Result				:= TRUE;
		END_IF;
	ELSE
		Internal.CTON_DB_On(IN := FALSE);
		Internal.CTON_DB_Off(IN := TRUE, PT := LREAL_TO_TIME(Par.FilterOffTime*1000.0));
		IF Internal.CTON_DB_Off.Q OR Par.FilterOffTime <= 0.0 THEN
			Signal.Result				:= FALSE;
		END_IF;
	END_IF;
//Edges
	IF EdgeReset THEN
		Signal.EdgePosResult			:= FALSE;
		Signal.EdgeNegResult			:= FALSE;
		Internal.StatusResult			:= FALSE;
	ELSE
		Signal.EdgeNegResult			:= FALSE;
		IF Internal.StatusResult AND NOT Signal.Result THEN
			Signal.EdgeNegResult		:= TRUE;
		END_IF;
		Signal.EdgePosResult			:= FALSE;
		IF NOT Internal.StatusResult AND Signal.Result THEN
			Signal.EdgePosResult		:= TRUE;
		END_IF;
		Internal.StatusResult 			:= Signal.Result;
	END_IF;
END_FUNCTION_BLOCK
```

### Library Logical/Libraries/TC_Recipe (IEC)
Depends on: MpBase, MpRecipe, AsBrStr, TC_General, TC_Str

#### Types.typ - Exported data types
```iecst
TYPE
	Recipe_Definition_typ : 	STRUCT
		MpLink : MpComIdentType;
		VarName : STRING[100];
		pVar : UDINT;
		SizeVar : UDINT;
		pCmpVar : UDINT;
		pDefaultVar : UDINT;
		DeviceName : STRING[50];
		FileName : STRING[255];
	END_STRUCT;
	TC_Recipe_Helper_Internal_typ : 	STRUCT
		MpRecipeRegPar_0 : MpRecipeRegPar;
		MpRecipeXml_0 : MpRecipeXml;
		LastState : TC_RECIPE_HELPER_STATE_ENUM;
		State : TC_RECIPE_HELPER_STATE_ENUM;
		ErrorReset : BOOL;
		CTON_Timeout : CTON;
	END_STRUCT;
	TC_RECIPE_HELPER_STATE_ENUM :
		(
		TC_RH_ST_RESET,
		TC_RH_ST_VALIDATE_INPUTS,
		TC_RH_ST_REG_PAR_W,
		TC_RH_ST_READY,
		TC_RH_ST_SAVE_W,
		TC_RH_ST_LOAD_W,
		TC_RH_ST_AUTO_LOAD_W,
		TC_RH_ST_AUTO_RESET_D,
		TC_RH_ST_AUTO_RESET_C,
		TC_RH_ST_AUTO_RESET_W,
		TC_RH_ST_AUTO_SAVE_W,
		TC_RH_ST_ERROR
		);
END_TYPE
```
